RTRIG_1(CLK :=INPUT_VAR.I_LOTBOX_DETECT_1);
RTRIG_2(CLK :=INPUT_VAR.I_LOTBOX_DETECT_2);
RTRIG_3(CLK :=INPUT_VAR.I_LOTBOX_DETECT_3);
RTRIG_4(CLK :=INPUT_VAR.I_LOTBOX_DETECT_4);
(*
IF RTRIG_1.Q THEN
	IF QUEUE_INDEX_1 =0  THEN
		QUEUE_INDEX_1 :=1;
	ELSIF QUEUE_INDEX_2 =0 THEN
		QUEUE_INDEX_2 :=1;
	ELSIF QUEUE_INDEX_3 =0 THEN
		QUEUE_INDEX_3 :=1;
	ELSIF QUEUE_INDEX_4 =0 THEN
		QUEUE_INDEX_4 :=1;
	END_IF	
	INPUT_VAR.O_LOTBOX_CLAMP_ON_1:=TRUE;
	INPUT_VAR.O_LOTBOX_CLAMP_OFF_1:=FALSE;
ELSIF RTRIG_2.Q THEN
	IF QUEUE_INDEX_1 =0  THEN
		QUEUE_INDEX_1 :=2;
	ELSIF QUEUE_INDEX_2 =0 THEN
		QUEUE_INDEX_2 :=2;
	ELSIF QUEUE_INDEX_3 =0 THEN
		QUEUE_INDEX_3 :=2;
	ELSIF QUEUE_INDEX_4 =0 THEN
		QUEUE_INDEX_4 :=2;
	END_IF
	INPUT_VAR.O_LOTBOX_CLAMP_ON_2:=TRUE;
	INPUT_VAR.O_LOTBOX_CLAMP_OFF_2:=FALSE;
ELSIF RTRIG_3.Q THEN
	IF QUEUE_INDEX_1 =0  THEN
		QUEUE_INDEX_1 :=3;
	ELSIF QUEUE_INDEX_2 =0 THEN
		QUEUE_INDEX_2 :=3;
	ELSIF QUEUE_INDEX_3 =0 THEN
		QUEUE_INDEX_3 :=3;
	ELSIF QUEUE_INDEX_4 =0 THEN
		QUEUE_INDEX_4 :=3;
	END_IF	
	INPUT_VAR.O_LOTBOX_CLAMP_ON_3:=TRUE;
	INPUT_VAR.O_LOTBOX_CLAMP_OFF_3:=FALSE;
ELSIF RTRIG_4.Q THEN
	IF QUEUE_INDEX_1 =0  THEN
		QUEUE_INDEX_1 :=4;
	ELSIF QUEUE_INDEX_2 =0 THEN
		QUEUE_INDEX_2 :=4;
	ELSIF QUEUE_INDEX_3 =0 THEN
		QUEUE_INDEX_3 :=4;
	ELSIF QUEUE_INDEX_4 =0 THEN
		QUEUE_INDEX_4 :=4;
	END_IF	
	INPUT_VAR.O_LOTBOX_CLAMP_ON_4:=TRUE;
	INPUT_VAR.O_LOTBOX_CLAMP_OFF_4:=FALSE;	
END_IF

IF NOT INPUT_VAR.I_LOTBOX_DETECT_1 THEN
	QUEUE_INDEX_1 :=0;
END_IF
IF NOT INPUT_VAR.I_LOTBOX_DETECT_2 THEN
	QUEUE_INDEX_2 :=0;
END_IF
IF NOT INPUT_VAR.I_LOTBOX_DETECT_3 THEN
	QUEUE_INDEX_3 :=0;
END_IF
IF NOT INPUT_VAR.I_LOTBOX_DETECT_4 THEN
	QUEUE_INDEX_4 :=0;
END_IF

IF INPUT_VAR.I_LOTEND THEN
	INPUT_VAR.O_LOTBOX_CLAMP_ON_1:=FALSE;
	INPUT_VAR.O_LOTBOX_CLAMP_ON_2:=FALSE;
	INPUT_VAR.O_LOTBOX_CLAMP_ON_3:=FALSE;
	INPUT_VAR.O_LOTBOX_CLAMP_ON_4:=FALSE;
	INPUT_VAR.O_LOTBOX_CLAMP_OFF_1:=TRUE;
	INPUT_VAR.O_LOTBOX_CLAMP_OFF_2:=TRUE;
	INPUT_VAR.O_LOTBOX_CLAMP_OFF_3:=TRUE;
	INPUT_VAR.O_LOTBOX_CLAMP_OFF_4:=TRUE;
			
END_IF
*)	
 
(*
INPUT_VAR.O_STOPPER_TRANSFER_A:=TMR11.Q ;
INPUT_VAR.O_STOPPER_TRANSFER_B:=TMR12.Q ;

TMR14(IN:=INPUT_G6_VAR.I_G6_END_FUKUDA,PT:=T#10S);
IF NOT TMR14.Q AND INPUT_G6_VAR.I_G6_END_FUKUDA THEN
	TMR11(IN:=FALSE);
	TMR12(IN:=FALSE);
ELSE
	TMR11(IN:=INPUT_VAR.I_FUKUDA_TRANSFER_AT_FRONT_A,PT:=T#2S);	
	TMR12(IN:=INPUT_VAR.I_FUKUDA_TRANSFER_AT_FRONT_B,PT:=T#2S);

END_IF
 

 IF INPUT_G6_VAR.I_G6_END_FUKUDA AND NOT INPUT_VAR.ACTIVE_PROGRAM_CHANGE THEN
	INPUT_VAR.ACTIVE_PROGRAM:=INPUT_VAR.ACTIVE_PROGRAM+1;
	IF INPUT_VAR.ACTIVE_PROGRAM=3 THEN
		INPUT_VAR.ACTIVE_PROGRAM:=1;
	END_IF
	INPUT_VAR.ACTIVE_PROGRAM_CHANGE:=TRUE;
 END_IF

 COUNTER_1(CU:=INPUT_G6_VAR.I_G6_END_CYCLE,RESET:=INPUT_G6_VAR.O_G6_START,PV:=14);
IF COUNTER_1.CV =1 THEN
	INPUT_VAR.ACTIVE_PROGRAM_CHANGE:=FALSE;
END_IF
 
*)
PULS1(IN:=NOT PULS2.Q,PT:=T#0.5S);
PULS2(IN:=PULS1.Q,PT:=T#0.5S);
IF INPUT_VAR.I_LOTBOX_DETECT_1 THEN
	INPUT_VAR.O_LOT_BOX_INDICATOR_1:=PULS1.Q;
	LOTBOX_TEMPI1:=1;
ELSE
	INPUT_VAR.O_LOT_BOX_INDICATOR_1:=FALSE;
	LOTBOX_TEMPI1:=0;
END_IF

IF INPUT_VAR.I_LOTBOX_DETECT_2 THEN
	INPUT_VAR.O_LOT_BOX_INDICATOR_2:=PULS1.Q;
	LOTBOX_TEMPI2:=1;
	ELSE
	LOTBOX_TEMPI2:=0;
	INPUT_VAR.O_LOT_BOX_INDICATOR_2:=FALSE;
END_IF

IF INPUT_VAR.I_LOTBOX_DETECT_3 THEN
	INPUT_VAR.O_LOT_BOX_INDICATOR_3:=PULS1.Q;
	LOTBOX_TEMPI3:=1;
	ELSE
	INPUT_VAR.O_LOT_BOX_INDICATOR_3:=FALSE;
	LOTBOX_TEMPI3:=0;
END_IF

IF INPUT_VAR.I_LOTBOX_DETECT_4 THEN
	INPUT_VAR.O_LOT_BOX_INDICATOR_4:=PULS1.Q;
	LOTBOX_TEMPI4:=1;
	ELSE
	INPUT_VAR.O_LOT_BOX_INDICATOR_4:=FALSE;
	LOTBOX_TEMPI4:=0;
END_IF
LOTBOX_ACCI:=LOTBOX_TEMPI1 +LOTBOX_TEMPI2+LOTBOX_TEMPI3+LOTBOX_TEMPI4;

//IF LOTBOX_ACCI >=3 THEN
IF INPUT_G6_VAR.I_G6_MOTORON AND INDEXING_2_VAR.I_INDEXING_2_HOME AND  LOADER_RS4_VAR.I_LOADER_RS4_MOTORON AND INDEXING_1_VAR.I_INDEXING_1_HOME AND SORTER_RS4_VAR.I_SORTER_RS4_MOTORON AND TESTER_C8_VAR.I_C8_MOTORON THEN
	INPUT_VAR.O_TOWER_LAMP_GREEN :=TRUE;
	INPUT_VAR.O_TOWER_LAMP_RED :=FALSE;
	
	SORTER_VAR.O_TOWER_LAMP_GREEN :=TRUE;
	SORTER_VAR.O_TOWER_LAMP_RED :=FALSE;
ELSE
	INPUT_VAR.O_TOWER_LAMP_RED :=TRUE;
	INPUT_VAR.O_TOWER_LAMP_GREEN :=FALSE;
	
	SORTER_VAR.O_TOWER_LAMP_GREEN :=FALSE;
	SORTER_VAR.O_TOWER_LAMP_RED :=TRUE;
END_IF
IF LOTBOX_ACCI =2 OR LOTBOX_ACCI =1 THEN
	INPUT_VAR.O_TOWER_LAMP_YELLOW :=PULS1.Q;
END_IF
IF INPUT_VAR.ALARM1 THEN
	INPUT_VAR.O_TOWER_LAMP_YELLOW :=PULS1.Q;
	SORTER_VAR.O_TOWER_LAMP_YELLOW :=PULS1.Q;
	//INPUT_VAR.O_TOWER_LAMP_BUZZER :=TRUE;
END_IF

END_PROGRAM

// ---- POUs/FUKUDA/LOAD_FUKUDA.TcPOU
PROGRAM LOAD_FUKUDA
VAR_INPUT

END_VAR

VAR
	TMR_DELAY: TON;
	TMR1:TON;
	TMR_STOPPER_A: TON;
	TMR_STOPPER_B: TON;
	I_FUKUDA_TRANSFER_AT_BACK_BTHEN: INT;
	TMR_ALARM: TON;
END_VAR

IF 	INPUT_VAR.TRANSPORT_IDX=0 AND 	INPUT_VAR.STATION_LOAD_IDX=0 AND 	INPUT_VAR.JIG_LOAD_IDX =0 THEN
	INPUT_VAR.TRANSPORT_IDX:=	INPUT_VAR.I_CURRENT_TRANSACTION.TRANSPORT_INDEX;
	INPUT_VAR.STATION_LOAD_IDX:=INPUT_VAR.I_CURRENT_TRANSACTION.STATION_NUMBER_LOAD;
	INPUT_VAR.JIG_LOAD_IDX :=	INPUT_VAR.I_CURRENT_TRANSACTION.JIG_INDEX_LOAD;
ELSE
CASE INPUT_VAR.I_CASE OF
0: //standby near lotbox
	IF INPUT_VAR.ACTIVE_ID=6 THEN
		INPUT_VAR.ACTIVE_ID:=1;
	END_IF
	
	INPUT_VAR.TRANSPORT_IDX:=	INPUT_VAR.I_CURRENT_TRANSACTION.TRANSPORT_INDEX;
	INPUT_VAR.STATION_LOAD_IDX:=INPUT_VAR.I_CURRENT_TRANSACTION.STATION_NUMBER_LOAD;
	INPUT_VAR.JIG_LOAD_IDX :=	INPUT_VAR.I_CURRENT_TRANSACTION.JIG_INDEX_LOAD;
	CASE INPUT_VAR.TRANSPORT_IDX OF
		2 : FUKUDA_MOVE(STEP_DATA_1:=INPUT_VAR.STATION_LOAD_IDX,
				STEP_DATA_2:=3,
				STEP_DATA_3:=INPUT_VAR.JIG_LOAD_IDX,
				STEP_DATA_4:=0,
				STEP_DATA_5:=1);
				INPUT_VAR.O_STOPPER_TRANSFER_B:=FALSE;
		1 : FUKUDA_MOVE(STEP_DATA_1:=INPUT_VAR.STATION_LOAD_IDX,
				STEP_DATA_2:=3,
				STEP_DATA_3:=INPUT_VAR.JIG_LOAD_IDX,
				STEP_DATA_4:=1,
				STEP_DATA_5:=0);
				INPUT_VAR.O_STOPPER_TRANSFER_A:=FALSE;
	END_CASE			
	input_var.O_VACUUM_On:=FALSE;
	input_var.O_VACUUM_OFF:=FALSE;	
			
1: //standby near lotbox
	
	IF INPUT_VAR.ACTIVE_ID=6 THEN
		INPUT_VAR.ACTIVE_ID:=1;
	END_IF
		FUKUDA_MOVE(STEP_DATA_1:=INPUT_VAR.STATION_LOAD_IDX,
				STEP_DATA_2:=4,
				STEP_DATA_3:=INPUT_VAR.JIG_LOAD_IDX,
				STEP_DATA_4:=0,
				STEP_DATA_5:=0);

		CASE INPUT_VAR.TRANSPORT_IDX OF
		1:
			INPUT_VAR.I_LOADING_DONE_A:=FALSE;
		
		2:
			INPUT_VAR.I_LOADING_DONE_B:=FALSE;
	END_CASE
	
				
2://vacuum position 
	IF INPUT_VAR.ACTIVE_ID=6 THEN
		INPUT_VAR.ACTIVE_ID:=1;
	END_IF
	INPUT_VAR.I_CASE:=INPUT_VAR.I_CASE+1;
	(*FUKUDA_MOVE(STEP_DATA_1:=INPUT_VAR.I_CURRENT_TRANSACTION.STATION_NUMBER_LOAD,
				STEP_DATA_2:=4,
				STEP_DATA_3:=INPUT_VAR.I_CURRENT_TRANSACTION.JIG_INDEX_LOAD,
				STEP_DATA_4:=0,
				STEP_DATA_5:=0);
	IF INPUT_VAR.ACTIVE_ID=3 THEN
		input_var.O_VACUUM_ON:=TRUE;
		input_var.O_VACUUM_OFF:=FALSE;	
	END_IF
	*)

3://vacuum position 
	IF INPUT_VAR.ACTIVE_ID=6 THEN
		INPUT_VAR.ACTIVE_ID:=1; 
	END_IF
	//INPUT_VAR.I_CASE:=INPUT_VAR.I_CASE+1;
	//IF INPUT_VAR.O_VACUUM_ON THEN
		FUKUDA_MOVE(STEP_DATA_1:=INPUT_VAR.STATION_LOAD_IDX,
				STEP_DATA_2:=4,
				STEP_DATA_3:=INPUT_VAR.JIG_LOAD_IDX,
				STEP_DATA_4:=0,
				STEP_DATA_5:=0);
	//ELSE
		
	//END_IF
4://vacuum position 
	IF INPUT_VAR.ACTIVE_ID=6 THEN
		INPUT_VAR.ACTIVE_ID:=1;
	END_IF
	input_var.O_VACUUM_ON:=TRUE; 
	input_var.O_VACUUM_OFF:=FALSE;
	 
	//CHECK JIG FUKUDA PRESENCE			
	IF  input_var.O_VACUUM_ON THEN
		TMR1(IN:=INPUT_VAR.I_VACUUM_ON,PT:=T#3S);
	END_IF
	IF TMR1.Q  AND INPUT_VAR.I_VACUUM_ON THEN
		input_var.O_VACUUM_ON:=FALSE;
		INPUT_VAR.JIG_FUKUDA_PRESENCE :=FALSE;
		INPUT_VAR.I_CASE:=10;
	ELSE
				INPUT_VAR.JIG_FUKUDA_PRESENCE :=TRUE;	
				FUKUDA_MOVE(STEP_DATA_1:=INPUT_VAR.STATION_LOAD_IDX,
				STEP_DATA_2:=2,
				STEP_DATA_3:=INPUT_VAR.JIG_LOAD_IDX,
				STEP_DATA_4:=0,
				STEP_DATA_5:=0);
	END_IF
				
		

5://vacuum position 
	IF INPUT_VAR.ACTIVE_ID=6 THEN
		INPUT_VAR.ACTIVE_ID:=1;
	END_IF
	
	FUKUDA_MOVE(STEP_DATA_1:=8,
				STEP_DATA_2:=2,
				STEP_DATA_3:=INPUT_VAR.JIG_LOAD_IDX,
				STEP_DATA_4:=0,
				STEP_DATA_5:=0);
	
6://gripping position
	IF INPUT_VAR.ACTIVE_ID=6 THEN
		INPUT_VAR.ACTIVE_ID:=1;
	END_IF

	FUKUDA_MOVE(STEP_DATA_1:=INPUT_VAR.TRANSPORT_IDX+4,
				STEP_DATA_2:=2,
				STEP_DATA_3:=12,
				STEP_DATA_4:=0,
				STEP_DATA_5:=0);


7://placing onto fukuda transport
	IF INPUT_VAR.ACTIVE_ID=6 THEN
		INPUT_VAR.ACTIVE_ID:=1;
	END_IF
	FUKUDA_MOVE(STEP_DATA_1:=INPUT_VAR.TRANSPORT_IDX+4,
				STEP_DATA_2:=2,
				STEP_DATA_3:=11,
				STEP_DATA_4:=0,
				STEP_DATA_5:=0);

8://placing onto fukuda transport
	IF INPUT_VAR.ACTIVE_ID=6 THEN
		INPUT_VAR.ACTIVE_ID:=1;
	END_IF
	
	FUKUDA_MOVE(STEP_DATA_1:=INPUT_VAR.TRANSPORT_IDX+4,
				STEP_DATA_2:=2,
				STEP_DATA_3:=11,
				STEP_DATA_4:=0,
				STEP_DATA_5:=0);
	(*IF INPUT_VAR.ACTIVE_ID=3 THEN
		input_var.O_VACUUM_On:=FALSE;
		input_var.O_VACUUM_OFF:=TRUE;	
	END_IF
	*)
	
9://homing
	IF INPUT_VAR.ACTIVE_ID=6 THEN
		INPUT_VAR.ACTIVE_ID:=1;
	END_IF
	IF INPUT_VAR.I_VACUUM_ON THEN
		FUKUDA_MOVE(STEP_DATA_1:=INPUT_VAR.TRANSPORT_IDX+4,
				STEP_DATA_2:=1,
				STEP_DATA_3:=13,//11
				STEP_DATA_4:=0,
				STEP_DATA_5:=0);
	ELSE
		input_var.O_VACUUM_On:=FALSE;
		input_var.O_VACUUM_OFF:=TRUE;
	END_IF	
				
10://pusH fukuda transport
	IF INPUT_VAR.ACTIVE_ID=6 THEN
		INPUT_VAR.ACTIVE_ID:=1;
	END_IF
	input_var.O_VACUUM_On:=FALSE;
	input_var.O_VACUUM_OFF:=TRUE;
	CASE INPUT_VAR.TRANSPORT_IDX OF
		2 :
			//IF NOT INPUT_VAR.I_FUKUDA_TRANSFER_AT_FRONT_B   THEN
				FUKUDA_MOVE(STEP_DATA_1:=0,
				STEP_DATA_2:=0,
				STEP_DATA_3:=0,
				STEP_DATA_4:=0,
				STEP_DATA_5:=2);
			//END_IF
				 
		1 : 
			//IF NOT INPUT_VAR.I_FUKUDA_TRANSFER_AT_FRONT_A  THEN
				FUKUDA_MOVE(STEP_DATA_1:=0,
				STEP_DATA_2:=0,
				STEP_DATA_3:=0,
				STEP_DATA_4:=2,
				STEP_DATA_5:=0);
			//END_IF
	END_CASE			 
11:
		input_var.O_VACUUM_On:=FALSE;
		input_var.O_VACUUM_OFF:=FALSE;
		CASE INPUT_VAR.TRANSPORT_IDX OF
		1:	
			TMR_ALARM(IN:= NOT INPUT_VAR.I_FUKUDA_TRANSFER_AT_FRONT_A,PT:=T#50S);
			IF INPUT_VAR.I_FUKUDA_TRANSFER_AT_FRONT_A THEN
				TMR_STOPPER_A(IN:=TRUE,PT:=T#0.8S);
				IF TMR_STOPPER_A.Q THEN 
					TMR_ALARM(IN:=FALSE);
					INPUT_VAR.O_STOPPER_TRANSFER_A:=TRUE;
					INPUT_VAR.I_LOADING_DONE_A:=TRUE;
					TMR1(IN:=FALSE);
					TMR_DELAY(IN:=FALSE);
					input_var.O_VACUUM_On:=FALSE;
					input_var.O_VACUUM_OFF:=TRUE;
					FLAG_VAR.ALLOW_EXECUTE_LOAD_FUKUDA:=FALSE;
					INPUT_G6_VAR.I_G6_ENABLE:=TRUE;
					INPUT_VAR.I_CASE:=100;
				END_IF
				
			ELSE
				TMR_STOPPER_A(IN:=FALSE);
				FUKUDA_MOVE(STEP_DATA_1:=0,
				STEP_DATA_2:=0,
				STEP_DATA_3:=0,
				STEP_DATA_4:=2,
				STEP_DATA_5:=0);
			END_IF 
			
			2:
				TMR_ALARM(IN:= NOT INPUT_VAR.I_FUKUDA_TRANSFER_AT_FRONT_B,PT:=T#50S);
			IF INPUT_VAR.I_FUKUDA_TRANSFER_AT_FRONT_B THEN
				
				TMR_STOPPER_B(IN:=TRUE,PT:=T#0.8S);
				IF TMR_STOPPER_B.Q THEN
					TMR_ALARM(IN:=FALSE);
					INPUT_VAR.O_STOPPER_TRANSFER_B:=TRUE;	
					INPUT_VAR.I_LOADING_DONE_B:=TRUE;
					TMR1(IN:=FALSE);
					TMR_DELAY(IN:=FALSE);
					input_var.O_VACUUM_On:=FALSE;
					input_var.O_VACUUM_OFF:=TRUE;
					FLAG_VAR.ALLOW_EXECUTE_LOAD_FUKUDA:=FALSE;
					INPUT_G6_VAR.I_G6_ENABLE:=TRUE;
					INPUT_VAR.I_CASE:=100;
				END_IF
			ELSE
				TMR_STOPPER_B(IN:=FALSE);
				FUKUDA_MOVE(STEP_DATA_1:=0,
				STEP_DATA_2:=0,
				STEP_DATA_3:=0,
				STEP_DATA_4:=0,
				STEP_DATA_5:=2);
			END_IF
			
	END_CASE 
	IF TMR_ALARM.Q THEN
					INPUT_VAR.I_LOADING_DONE_B:=FALSE;
					TMR1(IN:=FALSE);
					TMR_DELAY(IN:=FALSE);
					input_var.O_VACUUM_On:=FALSE;
					input_var.O_VACUUM_OFF:=FALSE;
					FLAG_VAR.ALLOW_EXECUTE_LOAD_FUKUDA:=FALSE;
					INPUT_VAR.I_CASE:=100;
	END_IF
100:
	
	FLAG_VAR.ALLOW_EXECUTE_LOAD_FUKUDA:=FALSE;								
								
END_CASE 
END_IF

END_PROGRAM

// ---- POUs/FUKUDA/RETURN_FUKUDA.TcPOU
PROGRAM RETURN_FUKUDA
VAR_INPUT

END_VAR

VAR
	TMR_DELAY: TON;
END_VAR

IF 	INPUT_VAR.TRANSPORT_IDX=0 AND 	INPUT_VAR.STATION_RETURN_IDX=0 AND 	INPUT_VAR.JIG_RETURN_IDX =0 THEN
	INPUT_VAR.TRANSPORT_IDX:=	INPUT_VAR.I_CURRENT_TRANSACTION.TRANSPORT_INDEX;
	INPUT_VAR.STATION_RETURN_IDX:=INPUT_VAR.I_CURRENT_TRANSACTION.STATION_NUMBER_RETURN;
	INPUT_VAR.JIG_RETURN_IDX :=	INPUT_VAR.I_CURRENT_TRANSACTION.JIG_INDEX_RETURN;
ELSE
CASE INPUT_VAR.I_CASE OF
0: //standby near lotbox
	IF INPUT_VAR.ACTIVE_ID=6 THEN
		INPUT_VAR.ACTIVE_ID:=1;
	END_IF
	
	INPUT_VAR.TRANSPORT_IDX:=	INPUT_VAR.I_CURRENT_TRANSACTION.TRANSPORT_INDEX;
	INPUT_VAR.STATION_RETURN_IDX:=INPUT_VAR.I_CURRENT_TRANSACTION.STATION_NUMBER_RETURN;
	INPUT_VAR.JIG_RETURN_IDX :=	INPUT_VAR.I_CURRENT_TRANSACTION.JIG_INDEX_RETURN;

	CASE INPUT_VAR.TRANSPORT_IDX OF
		2 : 
			INPUT_VAR.O_STOPPER_TRANSFER_B:=FALSE;			
			FUKUDA_MOVE(STEP_DATA_1:=3,
				STEP_DATA_2:=1,
				STEP_DATA_3:=12,
				STEP_DATA_4:=0,
				STEP_DATA_5:=1);
				INPUT_VAR.O_STOPPER_TRANSFER_B:=FALSE;
		1 : 
			INPUT_VAR.O_STOPPER_TRANSFER_A:=FALSE;
			FUKUDA_MOVE(STEP_DATA_1:=3,
				STEP_DATA_2:=1,
				STEP_DATA_3:=12,
				STEP_DATA_4:=1,
				STEP_DATA_5:=0);
				INPUT_VAR.O_STOPPER_TRANSFER_A:=FALSE;
	END_CASE			
	input_var.O_VACUUM_On:=FALSE;
	input_var.O_VACUUM_OFF:=FALSE;	
	TMR_DELAY(IN:=FALSE);

1://ready for picking up
	IF INPUT_VAR.ACTIVE_ID=6 THEN
		INPUT_VAR.ACTIVE_ID:=1;
	END_IF

		CASE INPUT_VAR.TRANSPORT_IDX OF
		1:
			INPUT_VAR.I_RETURN_DONE_A:=FALSE;
		
		2:
			INPUT_VAR.I_RETURN_DONE_B:=FALSE;
	END_CASE
	FUKUDA_MOVE(STEP_DATA_1:=3,
				STEP_DATA_2:=1,
				STEP_DATA_3:=13,
				STEP_DATA_4:=0,
				STEP_DATA_5:=0);	
			
2://ready for picking up
	IF INPUT_VAR.ACTIVE_ID=6 THEN
		INPUT_VAR.ACTIVE_ID:=1;
	END_IF

	CASE INPUT_VAR.TRANSPORT_IDX OF
	1:		
		IF INPUT_VAR.I_FUKUDA_TRANSFER_AT_BACK_A THEN
		FUKUDA_MOVE(STEP_DATA_1:=INPUT_VAR.TRANSPORT_IDX+4,
				STEP_DATA_2:=1,
				STEP_DATA_3:=11,
				STEP_DATA_4:=0,
				STEP_DATA_5:=0);
		END_IF
	2:
		IF INPUT_VAR.I_FUKUDA_TRANSFER_AT_BACK_B THEN
		FUKUDA_MOVE(STEP_DATA_1:=INPUT_VAR.TRANSPORT_IDX+4,
				STEP_DATA_2:=1,
				STEP_DATA_3:=11,
				STEP_DATA_4:=0,
				STEP_DATA_5:=0);
	END_IF
	END_CASE
	
		
3://placing onto fukuda transport
	IF INPUT_VAR.ACTIVE_ID=6 THEN
		INPUT_VAR.ACTIVE_ID:=1;
	END_IF

	FUKUDA_MOVE(STEP_DATA_1:=INPUT_VAR.TRANSPORT_IDX+4,
				STEP_DATA_2:=2,
				STEP_DATA_3:=11,
				STEP_DATA_4:=0,
				STEP_DATA_5:=0);
	
4://ready for picking up
	IF INPUT_VAR.ACTIVE_ID=6 THEN
		INPUT_VAR.ACTIVE_ID:=1;
	END_IF
	
	FUKUDA_MOVE(STEP_DATA_1:=INPUT_VAR.TRANSPORT_IDX+4,
				STEP_DATA_2:=6,
				STEP_DATA_3:=11,
				STEP_DATA_4:=0,
				STEP_DATA_5:=0);

5://gripping position
	IF INPUT_VAR.ACTIVE_ID=6 THEN
		INPUT_VAR.ACTIVE_ID:=1;
	END_IF
	
	IF NOT input_var.I_VACUUM_On THEN
		FUKUDA_MOVE(STEP_DATA_1:=INPUT_VAR.TRANSPORT_IDX+4,
				STEP_DATA_2:=2,
				STEP_DATA_3:=12,
				STEP_DATA_4:=0,
				STEP_DATA_5:=0);
	ELSE
		input_var.O_VACUUM_On:=TRUE;
		input_var.O_VACUUM_OFF:=FALSE;
	END_IF
	
				
6://vacuum position 
	IF INPUT_VAR.ACTIVE_ID=6 THEN
		INPUT_VAR.ACTIVE_ID:=1;
	END_IF
	
	FUKUDA_MOVE(STEP_DATA_1:=INPUT_VAR.STATION_RETURN_IDX,
				STEP_DATA_2:=3,
				STEP_DATA_3:=INPUT_VAR.JIG_RETURN_IDX,
				STEP_DATA_4:=0,
				STEP_DATA_5:=0);
				
7://vacuum position 
	IF INPUT_VAR.ACTIVE_ID=6 THEN
		INPUT_VAR.ACTIVE_ID:=1;
	END_IF
	TMR_DELAY(IN:=TRUE,PT:=T#1S);
	IF TMR_DELAY.Q THEN
			FUKUDA_MOVE(STEP_DATA_1:=INPUT_VAR.STATION_RETURN_IDX,
				STEP_DATA_2:=3,
				STEP_DATA_3:=14,
				STEP_DATA_4:=0,
				STEP_DATA_5:=0);
	END_IF
				
8://vacuum position 
	IF INPUT_VAR.ACTIVE_ID=6 THEN
		INPUT_VAR.ACTIVE_ID:=1;
	END_IF
	TMR_DELAY(IN:=FALSE);
	FUKUDA_MOVE(STEP_DATA_1:=INPUT_VAR.STATION_RETURN_IDX,
				STEP_DATA_2:=7,
				STEP_DATA_3:=16,
				STEP_DATA_4:=0,
				STEP_DATA_5:=0);
				
9://vacuum position 
	IF INPUT_VAR.ACTIVE_ID=6 THEN
		INPUT_VAR.ACTIVE_ID:=1;
	END_IF
	
	FUKUDA_MOVE(STEP_DATA_1:=INPUT_VAR.STATION_RETURN_IDX,
				STEP_DATA_2:=8,
				STEP_DATA_3:=INPUT_VAR.JIG_RETURN_IDX,
				STEP_DATA_4:=0,
				STEP_DATA_5:=0);
10: //standby near lotbox
	
	IF INPUT_VAR.ACTIVE_ID=6 THEN
		INPUT_VAR.ACTIVE_ID:=1;
	END_IF

	IF input_var.I_VACUUM_ON THEN
		FUKUDA_MOVE(STEP_DATA_1:=INPUT_VAR.STATION_RETURN_IDX,
				STEP_DATA_2:=4,
				STEP_DATA_3:=INPUT_VAR.JIG_RETURN_IDX,
				STEP_DATA_4:=0,
				STEP_DATA_5:=0);
	ELSE
		input_var.O_VACUUM_ON:=FALSE;
		input_var.O_VACUUM_OFF:=TRUE;			
	END_IF
	
				
11://vacuum position 
	IF INPUT_VAR.ACTIVE_ID=6 THEN
		INPUT_VAR.ACTIVE_ID:=1;
	END_IF
	FUKUDA_MOVE(STEP_DATA_1:=INPUT_VAR.STATION_RETURN_IDX,
				STEP_DATA_2:=1,
				STEP_DATA_3:=INPUT_VAR.JIG_RETURN_IDX,
				STEP_DATA_4:=0,
				STEP_DATA_5:=0);
	IF INPUT_VAR.ACTIVE_ID=3 THEN
		input_var.O_VACUUM_ON:=FALSE;
		input_var.O_VACUUM_OFF:=FALSE;	
	END_IF
	
12://vacuum position 
	IF INPUT_VAR.ACTIVE_ID=6 THEN
		INPUT_VAR.ACTIVE_ID:=1;
	END_IF
	FUKUDA_MOVE(STEP_DATA_1:=0,
				STEP_DATA_2:=1,
				STEP_DATA_3:=4,
				STEP_DATA_4:=0,
				STEP_DATA_5:=0);				
		
100:
	
	input_var.O_VACUUM_On:=FALSE;
	input_var.O_VACUUM_OFF:=FALSE;
END_CASE 
END_IF
IF INPUT_VAR.I_CASE=13 THEN
			CASE INPUT_VAR.TRANSPORT_IDX OF
		1:
			INPUT_VAR.I_RETURN_DONE_A:=TRUE;
		
		2:
			INPUT_VAR.I_RETURN_DONE_B:=TRUE;
	END_CASE
	IF INPUT_VAR.I_RETURN_DONE_A OR INPUT_VAR.I_RETURN_DONE_B THEN
		FLAG_VAR.ALLOW_EXECUTE_RETURN_FUKUDA:=FALSE;
		INPUT_VAR.I_CASE:=100;
	END_IF
END_IF

END_PROGRAM

// ---- POUs/FUKUDA/LOAD_FUKUDA_1.TcPOU
PROGRAM LOAD_FUKUDA_1
VAR_INPUT

END_VAR

VAR
	TMR_DELAY: TON;
	TMR1:TON;
END_VAR

CASE INPUT_VAR.I_CASE OF
0: //standby near lotbox
	IF INPUT_VAR.ACTIVE_ID=6 THEN
		INPUT_VAR.ACTIVE_ID:=1;
	END_IF
	CASE INPUT_VAR.I_CURRENT_TRANSACTION.TRANSPORT_INDEX OF
		2 : FUKUDA_MOVE(STEP_DATA_1:=INPUT_VAR.I_CURRENT_TRANSACTION.STATION_NUMBER_LOAD,
				STEP_DATA_2:=3,
				STEP_DATA_3:=INPUT_VAR.I_CURRENT_TRANSACTION.JIG_INDEX_LOAD,
				STEP_DATA_4:=0,
				STEP_DATA_5:=1);
		1 : FUKUDA_MOVE(STEP_DATA_1:=INPUT_VAR.I_CURRENT_TRANSACTION.STATION_NUMBER_LOAD,
				STEP_DATA_2:=3,
				STEP_DATA_3:=INPUT_VAR.I_CURRENT_TRANSACTION.JIG_INDEX_LOAD,
				STEP_DATA_4:=1,
				STEP_DATA_5:=0);
				
	input_var.O_VACUUM_On:=FALSE;
	input_var.O_VACUUM_OFF:=FALSE;	
	TMR_DELAY(IN:=FALSE);

	END_CASE
				
1: //standby near lotbox
	
	IF INPUT_VAR.ACTIVE_ID=6 THEN
		INPUT_VAR.ACTIVE_ID:=1;
	END_IF
		FUKUDA_MOVE(STEP_DATA_1:=INPUT_VAR.I_CURRENT_TRANSACTION.STATION_NUMBER_LOAD,
				STEP_DATA_2:=4,
				STEP_DATA_3:=INPUT_VAR.I_CURRENT_TRANSACTION.JIG_INDEX_LOAD,
				STEP_DATA_4:=0,
				STEP_DATA_5:=0);

		CASE INPUT_VAR.I_CURRENT_TRANSACTION.TRANSPORT_INDEX OF
		1:
			INPUT_VAR.I_LOADING_DONE_A:=FALSE;
		
		2:
			INPUT_VAR.I_LOADING_DONE_B:=FALSE;
	END_CASE

		
				
2://vacuum position 
	IF INPUT_VAR.ACTIVE_ID=6 THEN
		INPUT_VAR.ACTIVE_ID:=1;
	END_IF
	FUKUDA_MOVE(STEP_DATA_1:=INPUT_VAR.I_CURRENT_TRANSACTION.STATION_NUMBER_LOAD,
				STEP_DATA_2:=4,
				STEP_DATA_3:=INPUT_VAR.I_CURRENT_TRANSACTION.JIG_INDEX_LOAD,
				STEP_DATA_4:=0,
				STEP_DATA_5:=0);
	IF INPUT_VAR.ACTIVE_ID=3 THEN
		input_var.O_VACUUM_ON:=TRUE;
		input_var.O_VACUUM_OFF:=FALSE;	
	END_IF

3://vacuum position 
	IF INPUT_VAR.ACTIVE_ID=6 THEN
		INPUT_VAR.ACTIVE_ID:=1; 
	END_IF
	FUKUDA_MOVE(STEP_DATA_1:=INPUT_VAR.I_CURRENT_TRANSACTION.STATION_NUMBER_LOAD,
				STEP_DATA_2:=4,
				STEP_DATA_3:=INPUT_VAR.I_CURRENT_TRANSACTION.JIG_INDEX_LOAD,
				STEP_DATA_4:=0,
				STEP_DATA_5:=0);
	
 		
//CHECK JIG FUKUDA PRESENCE			
	IF  input_var.O_VACUUM_ON THEN
		TMR1(IN:=TRUE,PT:=T#2S);
		IF TMR1.Q THEN
			IF NOT INPUT_VAR.I_VACUUM_ON AND input_var.O_VACUUM_ON THEN
				INPUT_VAR.JIG_FUKUDA_PRESENCE :=TRUE;
			ELSE
				INPUT_VAR.JIG_FUKUDA_PRESENCE :=FALSE;	
				FUKUDA_MOVE(STEP_DATA_1:=INPUT_VAR.I_CURRENT_TRANSACTION.STATION_NUMBER_LOAD,
				STEP_DATA_2:=2,
				STEP_DATA_3:=INPUT_VAR.I_CURRENT_TRANSACTION.JIG_INDEX_LOAD,
				STEP_DATA_4:=0,
				STEP_DATA_5:=0);
				
				FUKUDA_MOVE(STEP_DATA_1:=INPUT_VAR.I_CURRENT_TRANSACTION.STATION_NUMBER_LOAD,
				STEP_DATA_2:=1,
				STEP_DATA_3:=INPUT_VAR.I_CURRENT_TRANSACTION.JIG_INDEX_LOAD,
				STEP_DATA_4:=0,
				STEP_DATA_5:=0);
			input_var.O_VACUUM_ON:=FALSE;
			input_var.O_VACUUM_OFF:=FALSE;
			TMR_DELAY(IN:=TRUE,PT:=T#2.5S);
		
			IF TMR_DELAY.Q THEN
				FLAG_VAR.ALLOW_EXECUTE_LOAD_FUKUDA:=FALSE;
				INPUT_VAR.I_CURRENT_TRANSACTION.JIG_INDEX_LOAD:=INPUT_VAR.I_CURRENT_TRANSACTION.JIG_INDEX_LOAD+0;
				INPUT_VAR.I_CASE:=0;
			END_IF
		END_IF
	ELSE
		TMR1(IN:=FALSE);	
	END_IF 
		
				//INPUT_VAR.JIG_FUKUDA_PRESENCE :=TRUE;
				//IF INPUT_VAR.I_CURRENT_TRANSACTION.JIG_INDEX_LOAD >=11 THEN
					//INPUT_VAR.I_CASE:=100;
			
				//FLAG_VAR.ALLOW_EXECUTE_LOAD_FUKUDA:=FALSE;
				//INPUT_VAR.I_CASE:=0;
				//INPUT_VAR.I_CURRENT_TRANSACTION.JIG_INDEX_LOAD:=1 ;
					//ELSE
						
				//END_IF
				
				//TMR_DELAY(IN:=FALSE);
				//LOAD_FUKUDA();
				//FLAG_VAR.ALLOW_EXECUTE_LOAD_FUKUDA:=FALSE;
	
	END_IF
 
	
4://vacuum position 
	IF INPUT_VAR.ACTIVE_ID=6 THEN
		INPUT_VAR.ACTIVE_ID:=1;
	END_IF
	
	FUKUDA_MOVE(STEP_DATA_1:=7,
				STEP_DATA_2:=4,
				STEP_DATA_3:=INPUT_VAR.I_CURRENT_TRANSACTION.JIG_INDEX_LOAD,
				STEP_DATA_4:=0,
				STEP_DATA_5:=0);
				

5://vacuum position 
	IF INPUT_VAR.ACTIVE_ID=6 THEN
		INPUT_VAR.ACTIVE_ID:=1;
	END_IF
	
	FUKUDA_MOVE(STEP_DATA_1:=8,
				STEP_DATA_2:=2,
				STEP_DATA_3:=INPUT_VAR.I_CURRENT_TRANSACTION.JIG_INDEX_LOAD,
				STEP_DATA_4:=0,
				STEP_DATA_5:=0);
	
6://gripping position
	IF INPUT_VAR.ACTIVE_ID=6 THEN
		INPUT_VAR.ACTIVE_ID:=1;
	END_IF

	FUKUDA_MOVE(STEP_DATA_1:=INPUT_VAR.I_CURRENT_TRANSACTION.TRANSPORT_INDEX+4,
				STEP_DATA_2:=2,
				STEP_DATA_3:=12,
				STEP_DATA_4:=0,
				STEP_DATA_5:=0);


7://placing onto fukuda transport
	IF INPUT_VAR.ACTIVE_ID=6 THEN
		INPUT_VAR.ACTIVE_ID:=1;
	END_IF
	FUKUDA_MOVE(STEP_DATA_1:=INPUT_VAR.I_CURRENT_TRANSACTION.TRANSPORT_INDEX+4,
				STEP_DATA_2:=2,
				STEP_DATA_3:=11,
				STEP_DATA_4:=0,
				STEP_DATA_5:=0);

8://placing onto fukuda transport
	IF INPUT_VAR.ACTIVE_ID=6 THEN
		INPUT_VAR.ACTIVE_ID:=1;
	END_IF
	
	FUKUDA_MOVE(STEP_DATA_1:=INPUT_VAR.I_CURRENT_TRANSACTION.TRANSPORT_INDEX+4,
				STEP_DATA_2:=2,
				STEP_DATA_3:=11,
				STEP_DATA_4:=0,
				STEP_DATA_5:=0);
	IF INPUT_VAR.ACTIVE_ID=3 THEN
		input_var.O_VACUUM_On:=FALSE;
		input_var.O_VACUUM_OFF:=TRUE;	
	END_IF

	
9://homing
	IF INPUT_VAR.ACTIVE_ID=6 THEN
		INPUT_VAR.ACTIVE_ID:=1;
	END_IF
	
	FUKUDA_MOVE(STEP_DATA_1:=INPUT_VAR.I_CURRENT_TRANSACTION.TRANSPORT_INDEX+4,
				STEP_DATA_2:=1,
				STEP_DATA_3:=11,
				STEP_DATA_4:=0,
				STEP_DATA_5:=0);
			
				
10://pusH fukuda transport
	IF INPUT_VAR.ACTIVE_ID=6 THEN
		INPUT_VAR.ACTIVE_ID:=1;
	END_IF
	input_var.O_VACUUM_OFF:=FALSE;
	CASE INPUT_VAR.I_CURRENT_TRANSACTION.TRANSPORT_INDEX OF
		2 : FUKUDA_MOVE(STEP_DATA_1:=0,
				STEP_DATA_2:=0,
				STEP_DATA_3:=0,
				STEP_DATA_4:=0,
				STEP_DATA_5:=2);
		1 : FUKUDA_MOVE(STEP_DATA_1:=0,
				STEP_DATA_2:=0,
				STEP_DATA_3:=0,
				STEP_DATA_4:=2,
				STEP_DATA_5:=0);
	END_CASE			 

100:

	input_var.O_VACUUM_On:=FALSE;
	input_var.O_VACUUM_OFF:=FALSE;	
	
END_CASE 
IF INPUT_VAR.I_CASE=11 THEN
			CASE INPUT_VAR.I_CURRENT_TRANSACTION.TRANSPORT_INDEX OF
		1:	
			IF INPUT_VAR.I_FUKUDA_TRANSFER_AT_FRONT_A THEN
				INPUT_VAR.I_LOADING_DONE_A:=TRUE;
				IF  INPUT_VAR.I_LOADING_DONE_A THEN
					FLAG_VAR.ALLOW_EXECUTE_LOAD_FUKUDA:=FALSE;			
					INPUT_VAR.I_CASE:=100;
				END_IF
			END_IF
			
				2:
			IF INPUT_VAR.I_FUKUDA_TRANSFER_AT_FRONT_B THEN
				INPUT_VAR.I_LOADING_DONE_B:=TRUE;
				IF  INPUT_VAR.I_LOADING_DONE_B THEN
					FLAG_VAR.ALLOW_EXECUTE_LOAD_FUKUDA:=FALSE;			
					INPUT_VAR.I_CASE:=100;
				END_IF
			END_IF
			
	END_CASE

END_IF

END_PROGRAM

// ---- POUs/LASER/LASER_MOVE.TcPOU
PROGRAM LASER_MOVE
//FUNCTION LASER_MOVE : BOOL
VAR_INPUT
	STEP_DATA_1: BYTE;
	STEP_DATA_2: BYTE;
	STEP_DATA_3: BYTE;
	STEP_DATA_4: BYTE;
	STEP_DATA_5: BYTE;

END_VAR

VAR
	
	(*
DataWordInput1 AT %IB232 : ARRAY [0..15] OF WORD; 
DataWordInput2 AT %IB264 : ARRAY [16..31] OF WORD;
DataWordInput3 AT %IB264 : ARRAY [32..47] OF WORD; 
DataWordInput4 AT %IB296 : ARRAY [48..56] OF WORD; 
DataWordOutput1 AT %QB232 : ARRAY [0..15] OF WORD; 
DataWordOutput2 AT %QB264 : ARRAY [16..31] OF WORD; 
DataWordOutput3 AT %QB296 : ARRAY [32..47] OF WORD; 
DataWordOutput4 AT %QB328 : ARRAY [48..56] OF WORD; 

DataWordInput1 AT %IB100 : ARRAY [0..15] OF WORD; 
DataWordInput2 AT %IB132 : ARRAY [16..31] OF WORD; 
DataWordInput3 AT %IB164 : ARRAY [32..47] OF WORD; 
DataWordInput4 AT %IB196 : ARRAY [48..56] OF WORD; 
DataWordOutput1 AT %QB100 : ARRAY [0..15] OF WORD; 
DataWordOutput2 AT %QB132 : ARRAY [16..31] OF WORD; 
DataWordOutput3 AT %QB164 : ARRAY [32..47] OF WORD; 
DataWordOutput4 AT %QB196 : ARRAY [48..56] OF WORD; 
	*)
	Gateway_Q0_MODE_COMMAND_0 AT %QX232.0 : BOOL ;
	Gateway_Q0_MODE_COMMAND_1 AT %QX232.1 : BOOL ;
	Gateway_Q0_RESET AT %QX232.4 : BOOL;
	Gateway_Q0_RESTART AT %QX232.5 : BOOL;
	Gateway_Q0_STOP AT %QX232.7 : BOOL;
	Gateway_Q1_0 AT %QX233.0 : BOOL;
	Gateway_Q1_1 AT %QX233.1 : BOOL;
	Gateway_Q1_2 AT %QX233.2 : BOOL;
	Gateway_Q1_3 AT %QX233.3 : BOOL;
	Gateway_Q1_4 AT %QX233.4 : BOOL;
	Gateway_Gateway_Unit_2_Status AT %QB234 : BYTE;
	Gateway_Q3_0 AT %QX235.0 : BOOL;
	Gateway_Q3_1 AT %QX235.1 : BOOL;
	Gateway_Q3_2 AT %QX235.2 : BOOL;
	Gateway_Q3_3 AT %QX235.3 : BOOL;	
	

	ID1_StepData AT %QB246 : BYTE;
	ID1_Hold AT %QX247.0 : BOOL;
	ID1_SVON AT %QX247.1 : BOOL;
	ID1_Drive AT %QX247.2 : BOOL;
	ID1_Reset AT %QX247.3 : BOOL;
	ID1_Setup AT %QX247.4 : BOOL;
	

	ID2_StepData AT %QB266 : BYTE;
	ID2_Hold AT %QX267.0 : BOOL;
	ID2_SVON AT %QX267.1 : BOOL;
	ID2_Drive AT %QX267.2 : BOOL;
	ID2_Reset AT %QX267.3 : BOOL;
	ID2_Setup AT %QX267.4 : BOOL;


	ID3_StepData AT %QB286 : BYTE;
	ID3_Hold AT %QX287.0 : BOOL;
	ID3_SVON AT %QX287.1 : BOOL;
	ID3_Drive AT %QX287.2 : BOOL;
	ID3_Reset AT %QX287.3 : BOOL;
	ID3_Setup AT %QX287.4 : BOOL;
	
	
	ID4_StepData AT %QB306 : BYTE;
	ID4_Hold AT %QX307.0 : BOOL;
	ID4_SVON AT %QX307.1 : BOOL;
	ID4_Drive AT %QX307.2 : BOOL;
	ID4_Reset AT %QX307.3 : BOOL;
	ID4_Setup AT %QX307.4 : BOOL;
	

	ID5_StepData AT %QB326 : BYTE;
	ID5_Hold AT %QX327.0 : BOOL;
	ID5_SVON AT %QX327.1 : BOOL;
	ID5_Drive AT %QX327.2 : BOOL;
	ID5_Reset AT %QX327.3 : BOOL;
	ID5_Setup AT %QX327.4 : BOOL;
	
	byte0 : BYTE;
	byte1 : BYTE;
	byte2 : BYTE;
	byte3 : BYTE;
	
	bit14_0 : BOOL;
	bit14_1 : BOOL;
	bit14_2 : BOOL;
	bit14_3 : BOOL;
	bit14_4 : BOOL;
	bit14_5 : BOOL;
	
	bit15_0 : BOOL;
	bit15_1 : BOOL;
	bit15_2 : BOOL;
	bit15_3 : BOOL;
	bit15_4 : BOOL; 
	
	bit34_0 : BOOL;
	bit34_1 : BOOL;
	bit34_2 : BOOL;
	bit34_3 : BOOL;
	bit34_4 : BOOL;
	bit34_5 : BOOL;
	
	bit35_0 : BOOL;
	bit35_1 : BOOL;
	bit35_2 : BOOL;
	bit35_3 : BOOL;
	bit35_4 : BOOL; 
	
	bit54_0 : BOOL;
	bit54_1 : BOOL;
	bit54_2 : BOOL;
	bit54_3 : BOOL;
	bit54_4 : BOOL;
	bit54_5 : BOOL;
	
	bit55_0 : BOOL;
	bit55_1 : BOOL;
	bit55_2 : BOOL;
	bit55_3 : BOOL;
	bit55_4 : BOOL; 
	
	bit74_0 : BOOL;
	bit74_1 : BOOL;
	bit74_2 : BOOL;
	bit74_3 : BOOL;
	bit74_4 : BOOL;
	bit74_5 : BOOL;
	
	bit75_0 : BOOL;
	bit75_1 : BOOL;
	bit75_2 : BOOL;
	bit75_3 : BOOL;
	bit75_4 : BOOL; 
	
	bit94_0 : BOOL;
	bit94_1 : BOOL;
	bit94_2 : BOOL;
	bit94_3 : BOOL;
	bit94_4 : BOOL;
	bit94_5 : BOOL;
	
	bit95_0 : BOOL;
	bit95_1 : BOOL;
	bit95_2 : BOOL;
	bit95_3 : BOOL;
	bit95_4 : BOOL; 	
	
	ID1_I0_MODE_COMMAND_0 AT %IX232.0 : BOOL :=0;
	ID1_I0_MODE_COMMAND_1 AT %IX232.1 : BOOL:=0;
	ID1_I0_READY AT %IX232.4 : BOOL;
	ID1_I0_ALARM AT %IX232.5 : BOOL;
	ID1_I0_INITIAL AT %IX232.6 : BOOL;
	ID1_I0_COMMUNICATING AT %IX232.7 : BOOL;
	ID1_I1_0 AT %IX233.0 : BOOL;
	ID1_I1_1 AT %IX233.1 : BOOL;
	ID1_I1_2 AT %IX233.2 : BOOL;
	ID1_I1_3 AT %IX233.3 : BOOL;
	ID1_I1_4 AT %IX233.4 : BOOL;
	ID1_I2_0 AT %IX234.0 : BOOL;
	ID1_I2_1 AT %IX234.1 : BOOL;
	ID1_I2_2 AT %IX234.2 : BOOL;
	ID1_I2_3 AT %IX234.3 : BOOL;
	ID1_I2_4 AT %IX234.4 : BOOL;

	ID1_I3_0 AT %IX235.0 : BOOL;
	ID1_I3_1 AT %IX235.1 : BOOL;
	
	ID1_I32_0 AT %IX264.0 : BOOL;
	ID1_I32_1 AT %IX264.1 : BOOL;
	ID1_I33_0 AT %IX265.0 : BOOL;
	ID1_I33_1 AT %IX265.1 : BOOL;
(*-----------------------------------------------------------*)

	iTest15: SINT;
	iTest16: SINT;
	
	bTest1 : BOOL;
	bTest2 : BOOL;
	bTest3 : BOOL;
	bTest4 : BOOL;
	bTest5 : BOOL;
	bTest6 : BOOL;
	bTest7 : BOOL;
	bTest8 : BOOL;
	bTest9 : BOOL;
	bTest10 : BOOL;
	bTest11 : BOOL;
	bTest12 : BOOL;
	bTest13 : BOOL;
	bTest14 : BOOL;
	
	StepData1 : BYTE;
	StepData2 : BYTE;
	StepData3 : BYTE;
	StepData4 : BYTE;
	StepData5 : BYTE;
	
	star :BOOL;
	hom : BOOL;

	reset: BOOL;
	
	ID1_ALARM AT%IX247.7 : BOOL;
	ID2_ALARM AT%IX267.7 : BOOL;
	ID3_ALARM AT%IX287.7 : BOOL;
	ID4_ALARM AT%IX307.7 : BOOL;
	ID5_ALARM AT%IX327.7 : BOOL;
	
	ID1_SVRE AT%IX247.1 : BOOL;
	ID2_SVRE AT%IX267.1 : BOOL;
	ID3_SVRE AT%IX287.1 : BOOL;
	ID4_SVRE AT%IX307.1 : BOOL;
	ID5_SVRE AT%IX327.1 : BOOL;
	
	ID1_INP AT%IX247.3 : BOOL;
	ID2_INP AT%IX267.3 : BOOL;
	ID3_INP AT%IX287.3 : BOOL;
	ID4_INP AT%IX307.3 : BOOL;
	ID5_INP AT%IX327.3 : BOOL;
	
	PROSES: STRING;
	STAGE: INT;
	
	PROCESS: INT;
	START_PROCESS: BOOL;
	STEP_DATAS: INT;
	PROCESS_DELAY: TIME :=T#300MS;
	LASER_RUNNING: BOOL :=FALSE;
	ACTIVE_STEPDATA : BYTE;
	//ACTIVE_ID: INT :=1;
	TMR1: TON;
	TMR2: TON;
	TMR3: TON;
	TMR4: TON;
	TMR5: TON;
	TMR6: TON;
	TMR10: Ton;
	TMR11: TON;
	TMR12: TON;
	TMR13: TON;
	TMR14: TON;
	TMR20: TON;
	TMR21: TON;
	TMR22: TON;
	TMR23: TON;
	TMR30: TON;
	TMR31: TON;
	TMR32: TON;
	TMR33: TON;
	TMR40: TON;
	TMR41: TON;
	TMR42: TON;
	TMR43: TON;
	TMR50: TON;
	TMR51: TON;
	TMR52: TON;
	TMR53: TON;
	
	
	TMR101: TON;
	TMR102: TON;
	TMR103: TON;
	TMR104: TON;
	TMR105: TON;
	TMR106: TON;
	ID5: INT;
	TMR7: Ton;
	TMR_RES_CARTSN: TOF;
	TMR_ACTIVATE_RESET: TON;
	TMR_RST: TON;
	TMR_RST1: TON;
	ID2_READY: BOOL;
	ID4_READY: BOOL;
	ID5_READY: BOOL;
END_VAR


PROCESS_DELAY:= T#400MS;
IF 	SORTER_VAR.ACTIVE_ID >=0 THEN
STEP_DATA_1:=STEP_DATA_1+1;

IF STEP_DATA_2>=5 THEN
	STEP_DATA_2:=STEP_DATA_2+1;
END_IF

STEP_DATA_3:=STEP_DATA_3+1;	
END_IF

IF NOT ID1_SVRE OR NOT ID2_SVRE OR NOT ID3_SVRE OR NOT ID4_SVRE OR NOT ID5_SVRE THEN
	TMR_RST(IN:=TRUE,PT:=T#10S);
	IF TMR_RST.Q THEN
		SORTER_VAR.O_RESET_CARTESSIAN:=TRUE;
		TMR_RST1(IN:=TRUE,PT:=T#1S);
		IF TMR_RST1.Q THEN
			SORTER_VAR.O_RESET_CARTESSIAN:=FALSE;
			TMR_RST(IN:=FALSE);
			TMR_RST1(IN:=FALSE);
			FLAG_VAR.ALLOW_EXECUTE_LOAD_LASER :=FALSE;
			FLAG_VAR.ALLOW_EXECUTE_RETURN_LASER:=FALSE;
			LASER_MOVE(STEP_DATA_1:=0,
				STEP_DATA_2:=0,
				STEP_DATA_3:=0,
				STEP_DATA_4:=0,
				STEP_DATA_5:=0);
		END_IF
	END_IF
ELSE
	SORTER_VAR.O_RESET_CARTESSIAN:=FALSE;
	TMR_RST(IN:=FALSE);
	TMR_RST1(IN:=FALSE);
END_IF
IF NOT SORTER_VAR.LASER_HOME THEN //LASER_running THEN
	IF  ID1_SVRE AND ID2_SVRE  AND  ID3_SVRE AND  ID4_SVRE AND  ID5_SVRE THEN
		TMR1(IN:=TRUE,PT:=T#0.5S);
		TMR4(IN:=TRUE,PT:=T#5S);
		TMR5(IN:=TRUE,PT:=T#5.5S);
		TMR6(IN:=TRUE,PT:=T#25S);
		
		IF ID2_SVRE THEN
			ID2_SETUP:=TRUE;
			IF ID2_INP THEN
				ID2_READY:=TRUE;
				IF ID3_SVRE THEN
					ID3_SETUP :=TRUE;
					IF ID3_INP THEN
						ID2_READY:=TRUE;
						IF ID1_SVRE THEN
							ID1_SETUP :=TRUE;
						ELSE
							ID1_SVON :=TRUE;	
						END_IF
					END_IF
				ELSE
					ID3_SVON :=TRUE;
				END_IF
			END_IF
		ELSE
			ID2_SVON :=TRUE;					
		END_IF
		(*
		IF ID1_SVRE THEN
			ID1_SETUP :=TMR5.Q;
		ELSE
			ID1_SVON :=TRUE;	
		END_IF

		IF ID2_SVRE THEN
			ID2_SETUP :=TMR1.Q;
		ELSE
			ID2_SVON :=TRUE;	
		END_IF
	
		IF ID3_SVRE THEN
		ID3_SETUP :=TMR4.Q;
		ELSE
			ID3_SVON :=TRUE;	
		END_IF
		*)
		CASE SORTER_VAR.I_CURRENT_TRANSACTION.TRANSPORT_INDEX OF
		1:
			TMR2(IN:=TRUE,PT:=T#1S);
			IF ID4_SVRE THEN
				ID4_SETUP :=TMR2.Q;
				IF ID4_INP THEN
					ID4_READY:=TRUE;
				END_IF
			ELSE
				ID4_SVON :=TRUE;	
			END_IF
		2:
			TMR3(IN:=TRUE,PT:=T#1.5S);
			IF ID5_SVRE THEN
				ID5_SETUP :=TMR3.Q;
				IF ID5_INP THEN
					ID5_READY:=TRUE;
				END_IF
			ELSE
				ID5_SVON :=TRUE;	
			END_IF
		END_CASE

	//IF TMR6.Q THEN
	IF ID1_INP AND ID2_INP AND ID3_INP AND (ID4_INP OR ID5_INP) THEN
		ID1_SETUP :=FALSE;
		ID2_SETUP :=FALSE;
		ID3_SETUP :=FALSE;
		ID4_SETUP :=FALSE;
		ID5_SETUP :=FALSE;
	
		TMR1(IN:=FALSE);
		TMR2(IN:=FALSE);
		TMR3(IN:=FALSE);
		TMR4(IN:=FALSE);
		TMR5(IN:=FALSE);
	//ACTIVE_ID:=1;
	//LASER_RUNNING:=TRUE;
		SORTER_VAR.LASER_HOME:=TRUE;
	END_IF
	
	ELSE
				
	ID1_SVON :=TRUE;
	ID2_SVON :=TRUE;
	ID3_SVON :=TRUE;
	ID4_SVON :=TRUE;
	ID5_SVON :=TRUE;

	END_IF
ELSE
	TMR6(IN:=FALSE);

	CASE SORTER_VAR.ACTIVE_ID OF
	0:
		//SORTER_VAR.I_LASER_RUNNING:=FALSE;
		SORTER_VAR.ACTIVE_ID:=6;
		IF 	FLAG_VAR.ALLOW_EXECUTE_LOAD_NG OR FLAG_VAR.ALLOW_EXECUTE_RETURN_NG THEN
			SORTER_VAR.I_NG_CASE:=SORTER_VAR.I_NG_CASE+1;
		ELSE
			SORTER_VAR.I_CASE:=SORTER_VAR.I_CASE+1;
		END_IF
	1:
		IF STEP_DATA_1 = 0 THEN
			SORTER_VAR.ACTIVE_ID:=2;
		ELSE
			IF ID1_ALARM THEN
				Reset := TRUE;
				TMR10(IN:=TRUE,PT:= PROCESS_DELAY);
				IF TMR10.Q THEN
					Reset := FALSE;
				END_IF
			ELSE
				ID1_StepData :=STEP_DATA_1;
				ID1_Drive := FALSE;
				TMR11(IN:=TRUE,PT:= PROCESS_DELAY);
				IF TMR11.Q THEN
					ID1_Drive := TRUE;
					TMR12(IN:=TMR11.Q,PT:= PROCESS_DELAY);
					IF TMR12.Q THEN
						
						IF ID1_INP THEN
							TMR10(IN:=FALSE);
						TMR11(IN:=FALSE);
						TMR12(IN:=FALSE);
						ID1_Drive := FALSE;
						SORTER_VAR.ACTIVE_ID:=2;
						SORTER_VAR.LASER_HOME:=TRUE;
						END_IF
					END_IF
				END_IF
			END_IF
		END_IF
	//	SORTER_VAR.I_CASE:=SORTER_VAR.I_CASE+1;
		//SORTER_VAR.I_LASER_RUNNING:=FALSE;
	2:
		IF STEP_DATA_2 = 0 THEN
			SORTER_VAR.ACTIVE_ID:=3;
		ELSE
			
			IF ID2_ALARM THEN
				Reset := TRUE;
				TMR20(IN:=TRUE,PT:= PROCESS_DELAY);
				IF TMR20.Q THEN
					Reset := FALSE;
				END_IF
			ELSE
			ID2_StepData :=STEP_DATA_2;
			TMR21(IN:=TRUE,PT:= PROCESS_DELAY);
			IF TMR21.Q THEN
				ID2_Drive := TRUE;
				TMR22(IN:=TMR21.Q,PT:= PROCESS_DELAY);
				IF TMR22.Q THEN
					
					IF ID2_INP THEN
						TMR20(IN:=FALSE);
					TMR21(IN:=FALSE);
					TMR22(IN:=FALSE);
					ID2_Drive := FALSE;
						SORTER_VAR.ACTIVE_ID:=3;
					END_IF
					END_IF
			END_IF
			END_IF
		END_IF
	3:
		IF STEP_DATA_3 = 0 THEN
			SORTER_VAR.ACTIVE_ID:=4;
		ELSE
			
		IF ID3_ALARM THEN
			Reset := TRUE;
			TMR30(IN:=START_PROCESS,PT:= PROCESS_DELAY);
			IF TMR30.Q THEN
				Reset := FALSE;
			END_IF
		ELSE
		
		ID3_StepData :=STEP_DATA_3;
		TMR31(IN:=TRUE,PT:= PROCESS_DELAY);
		IF TMR31.Q THEN
			
			ID3_DRIVE := TRUE;	
			TMR32(IN:=TMR31.Q,PT:= PROCESS_DELAY);
			
			IF TMR32.Q THEN
				
				IF ID3_INP THEN
				SORTER_VAR.ACTIVE_ID:=4;
ID3_Drive := FALSE;
				TMR30(IN:=FALSE);
				TMR31(IN:=FALSE);
				TMR32(IN:=FALSE);
				END_IF
			END_IF
		END_IF
		END_IF
	END_IF
4:
		IF STEP_DATA_4 = 0 THEN
			SORTER_VAR.ACTIVE_ID:=5;
		ELSE
			IF ID4_ALARM THEN
				Reset := TRUE;
				TMR40(IN:=TRUE,PT:= PROCESS_DELAY);
				IF TMR40.Q THEN
					Reset := FALSE;
				END_IF
			ELSE
			IF NOT ID4_READY THEN
				IF ID4_SVRE THEN
					ID4_SETUP :=TRUE;
					IF ID4_INP THEN
						ID4_READY:=TRUE;
					END_IF
				END_IF
			ELSE

			ID4_StepData :=STEP_DATA_4;
			TMR41(IN:=TRUE,PT:= PROCESS_DELAY);
			IF TMR41.Q THEN
				ID4_Drive := TRUE;
				TMR42(IN:=TMR41.Q,PT:= PROCESS_DELAY);
				
				IF TMR42.Q THEN
			
					IF ID4_INP THEN
						SORTER_VAR.ACTIVE_ID:=5;
								ID4_Drive := FALSE;
					TMR40(IN:=FALSE);
					TMR41(IN:=FALSE);
					TMR42(IN:=FALSE);
					END_IF
				END_IF
			END_IF
			END_IF
			END_IF
		END_IF
	5:
		IF STEP_DATA_5 = 0 THEN
			SORTER_VAR.ACTIVE_ID:=0;
		ELSE
			
			IF ID5_ALARM THEN
				Reset := TRUE;
				TMR50(IN:=TRUE,PT:= PROCESS_DELAY);
				IF TMR50.Q THEN
					Reset := FALSE;
				END_IF
			ELSE
				IF NOT ID5_READY THEN
				IF ID5_SVRE THEN
					ID5_SETUP :=TRUE;
					IF ID5_INP THEN
						ID5_READY:=TRUE;
					END_IF
				END_IF
			ELSE
			ID5_StepData :=STEP_DATA_5;
			TMR51(IN:=TRUE,PT:= PROCESS_DELAY);
			IF TMR51.Q THEN
				ID5_Drive := TRUE;	
				TMR52(IN:=TMR51.Q,PT:= PROCESS_DELAY);
				IF TMR52.Q THEN
					
					IF ID5_INP THEN
					SORTER_VAR.ACTIVE_ID:=0;
ID5_Drive := FALSE;
					TMR50(IN:=FALSE);
					TMR51(IN:=FALSE);
					TMR52(IN:=FALSE);
				END_IF
				END_IF
			END_IF
			END_IF
			END_IF
		END_IF
		
END_CASE 

	//START_PROCESS := FALSE;
END_IF
TMR7(IN:=reset,PT:= T#1S);
IF  tmr7.Q THEN
	reset:=FALSE;
END_IF
IF ID1_ALARM OR ID2_ALARM OR ID3_ALARM OR ID4_ALARM OR ID5_ALARM THEN
	reset:=TRUE;
	INPUT_VAR.ALARM1:=ID1_ALARM OR ID2_ALARM OR ID3_ALARM OR ID4_ALARM OR ID5_ALARM;
ELSE
	reset:=FALSE;
END_IF
IF reset THEN
	ID1_Reset := TRUE;
	ID2_Reset := TRUE;
	ID3_Reset := TRUE;
	ID4_Reset := TRUE;
	ID5_Reset := TRUE;
	TMR_ACTIVATE_RESET(IN:=TRUE,PT:=T#10S);
	IF TMR_ACTIVATE_RESET.Q THEN
		TMR_RES_CARTSN(IN:=TRUE,PT:=T#0.5S);
	END_IF
	
ELSE
	TMR_ACTIVATE_RESET(IN:=FALSE);
	TMR_RES_CARTSN(IN:=FALSE);
	ID1_Reset := FALSE;
	ID2_Reset := FALSE;
	ID3_Reset := FALSE;
	ID4_Reset := FALSE;
	ID5_Reset := FALSE;
END_IF
SORTER_VAR.O_RESET_CARTESSIAN := TMR_RES_CARTSN.Q;

END_PROGRAM

// ---- POUs/LASER/LASER_PROG.TcPOU
PROGRAM LASER_PROG
VAR
	
	PULS1: TON;
	PULS2: TON;
	CNT1: CTU;
	LOTBOX_ACC: INT;
	LOTBOX_ACC1: INT;
	LOTBOX_TEMP1: INT;
	LOTBOX_TEMP2: INT;
	LOTBOX_TEMP3: INT;
	LOTBOX_TEMP4: INT;
	NGBOX_TEMP: INT;
	NGBOX_TEMP1: INT;
	NGBOX_TEMP2: INT;
	NGBOX_TEMP3: INT;
	NGBOX_TEMP4: INT;
	NGBOX_ACC: INT;
END_VAR


PULS1(IN:=NOT PULS2.Q,PT:=T#0.5S);
PULS2(IN:=PULS1.Q,PT:=T#1S);
CNT1(CU:=PULS1.Q,RESET:=CNT1.Q,PV:=9);
(*
IF CNT1.CV=1 THEN
	SORTER_VAR.O_NG_BOX_INDICATOR_4:=TRUE;
END_IF
IF CNT1.CV=2 THEN
	SORTER_VAR.O_NG_BOX_INDICATOR_3:=TRUE;
END_IF
IF CNT1.CV=3 THEN
	SORTER_VAR.O_NG_BOX_INDICATOR_2:=TRUE;
END_IF
IF CNT1.CV=4 THEN
	SORTER_VAR.O_NG_BOX_INDICATOR_1:=TRUE;
END_IF
IF CNT1.CV=5 THEN
	SORTER_VAR.O_LOT_BOX_INDICATOR_4:=TRUE;
END_IF
IF CNT1.CV=6 THEN
	SORTER_VAR.O_LOT_BOX_INDICATOR_3:=TRUE;
END_IF
IF CNT1.CV=7 THEN
	SORTER_VAR.O_LOT_BOX_INDICATOR_2:=TRUE;
END_IF
IF CNT1.CV=8 THEN
	SORTER_VAR.O_LOT_BOX_INDICATOR_1:=TRUE;
END_IF
IF CNT1.Q THEN
	SORTER_VAR.O_LOT_BOX_INDICATOR_1:=FALSE;
	SORTER_VAR.O_LOT_BOX_INDICATOR_2:=FALSE;
	SORTER_VAR.O_LOT_BOX_INDICATOR_3:=FALSE;
	SORTER_VAR.O_LOT_BOX_INDICATOR_4:=FALSE;
	SORTER_VAR.O_NG_BOX_INDICATOR_1:=FALSE;
	SORTER_VAR.O_NG_BOX_INDICATOR_2:=FALSE;
	SORTER_VAR.O_NG_BOX_INDICATOR_3:=FALSE;
	SORTER_VAR.O_NG_BOX_INDICATOR_4:=FALSE;
END_IF
*)
IF SORTER_VAR.I_LOTBOX_DETECT_1 THEN
	SORTER_VAR.O_LOT_BOX_INDICATOR_1:=PULS1.Q;
	LOTBOX_TEMP1:=1;
ELSE
	SORTER_VAR.O_LOT_BOX_INDICATOR_1:=FALSE;
	LOTBOX_TEMP1:=0;
END_IF

IF SORTER_VAR.I_LOTBOX_DETECT_2 THEN
	SORTER_VAR.O_LOT_BOX_INDICATOR_2:=PULS1.Q;
	LOTBOX_TEMP2:=1;
	ELSE
	LOTBOX_TEMP2:=0;
	SORTER_VAR.O_LOT_BOX_INDICATOR_2:=FALSE;
END_IF

IF SORTER_VAR.I_LOTBOX_DETECT_3 THEN
	SORTER_VAR.O_LOT_BOX_INDICATOR_3:=PULS1.Q;
	LOTBOX_TEMP3:=1;
	ELSE
	SORTER_VAR.O_LOT_BOX_INDICATOR_3:=FALSE;
	LOTBOX_TEMP3:=0;
END_IF

IF SORTER_VAR.I_LOTBOX_DETECT_4 THEN
	SORTER_VAR.O_LOT_BOX_INDICATOR_4:=PULS1.Q;
	LOTBOX_TEMP4:=1;
	ELSE
	SORTER_VAR.O_LOT_BOX_INDICATOR_4:=FALSE;
	LOTBOX_TEMP4:=0;
END_IF
LOTBOX_ACC:=LOTBOX_TEMP1 +LOTBOX_TEMP2+LOTBOX_TEMP3+LOTBOX_TEMP4;

IF LOTBOX_ACC >=3 THEN
	//SORTER_VAR.O_TOWER_LAMP_BUZZER :=TRUE;
	ELSE
	SORTER_VAR.O_TOWER_LAMP_BUZZER :=FALSE;
END_IF

IF NOT SORTER_VAR.I_NG_BOX_DETECT_1 THEN
		SORTER_VAR.O_NG_BOX_INDICATOR_1:=PULS1.Q;
		NGBOX_TEMP1:=1;
		ELSE
		SORTER_VAR.O_NG_BOX_INDICATOR_1:=FALSE;
		NGBOX_TEMP1:=0;
END_IF

IF NOT SORTER_VAR.I_NG_BOX_DETECT_2 THEN
		SORTER_VAR.O_NG_BOX_INDICATOR_2:=PULS1.Q;
		NGBOX_TEMP2:=1;
		ELSE
		SORTER_VAR.O_NG_BOX_INDICATOR_2:=FALSE;
		NGBOX_TEMP2:=0;
END_IF

IF NOT SORTER_VAR.I_NG_BOX_DETECT_3 THEN
		SORTER_VAR.O_NG_BOX_INDICATOR_3:=PULS1.Q;
		NGBOX_TEMP3:=1;
		ELSE
		SORTER_VAR.O_NG_BOX_INDICATOR_3:=FALSE;
		NGBOX_TEMP3:=0;
END_IF

IF NOT SORTER_VAR.I_NG_BOX_DETECT_4 THEN
		SORTER_VAR.O_NG_BOX_INDICATOR_4:=PULS1.Q;
		NGBOX_TEMP4:=1;
		ELSE
		SORTER_VAR.O_NG_BOX_INDICATOR_4:=FALSE;
		NGBOX_TEMP4:=0;
END_IF
NGBOX_ACC:=NGBOX_TEMP1+NGBOX_TEMP2+NGBOX_TEMP3+NGBOX_TEMP4;
IF NGBOX_ACC >=3 THEN
	//SORTER_VAR.O_TOWER_LAMP_BUZZER :=TRUE;
	ELSE
	SORTER_VAR.O_TOWER_LAMP_BUZZER :=FALSE;
END_IF

END_PROGRAM

// ---- POUs/LASER/LOAD_LASER.TcPOU
PROGRAM LOAD_LASER
VAR_INPUT

END_VAR

VAR
	TMR_DELAY: TON;
	TMR1:TON;
	TMR_STOPPER_A: TON;
	TMR_STOPPER_B: TON;
	TMR_DLY: TON;
	TMR_DLY2: TON;

END_VAR

CASE SORTER_VAR.I_CASE OF
0: //standby near lotbox
	IF SORTER_VAR.ACTIVE_ID=6 THEN
		SORTER_VAR.ACTIVE_ID:=1;
	END_IF
	SORTER_VAR.TRANSPORT_IDX:=		SORTER_VAR.I_CURRENT_TRANSACTION.TRANSPORT_INDEX;
	SORTER_VAR.STATION_LOAD_IDX:=	SORTER_VAR.I_CURRENT_TRANSACTION.STATION_NUMBER_LOAD;
	SORTER_VAR.JIG_LOAD_IDX:=		SORTER_VAR.I_CURRENT_TRANSACTION.JIG_INDEX_LOAD;
	
	IF SORTER_VAR.TRANSPORT_IDX=0 AND SORTER_VAR.STATION_LOAD_IDX=0 AND SORTER_VAR.JIG_LOAD_IDX=0 THEN
		SORTER_VAR.TRANSPORT_IDX:=		SORTER_VAR.I_CURRENT_TRANSACTION.TRANSPORT_INDEX;
		SORTER_VAR.STATION_LOAD_IDX:=	SORTER_VAR.I_CURRENT_TRANSACTION.STATION_NUMBER_LOAD;
		SORTER_VAR.JIG_LOAD_IDX:=		SORTER_VAR.I_CURRENT_TRANSACTION.JIG_INDEX_LOAD;
	ELSE
		
	CASE SORTER_VAR.TRANSPORT_IDX OF
		2 : LASER_MOVE(STEP_DATA_1:=SORTER_VAR.STATION_LOAD_IDX,
				STEP_DATA_2:=0,
				STEP_DATA_3:=SORTER_VAR.JIG_LOAD_IDX,
				STEP_DATA_4:=0,
				STEP_DATA_5:=1);
				SORTER_VAR.O_STOPPER_TRANSFER_B:=FALSE;
				//SORTER_VAR.I_LOADING_DONE_B:=FALSE;
		1 : LASER_MOVE(STEP_DATA_1:=SORTER_VAR.STATION_LOAD_IDX,
				STEP_DATA_2:=0,
				STEP_DATA_3:=SORTER_VAR.JIG_LOAD_IDX,
				STEP_DATA_4:=1,
				STEP_DATA_5:=0);
				SORTER_VAR.O_STOPPER_TRANSFER_A:=FALSE;
				//SORTER_VAR.I_LOADING_DONE_A:=FALSE;
	END_CASE
END_IF			
	SORTER_VAR.O_VACUUM_On:=FALSE;
	SORTER_VAR.O_VACUUM_OFF:=FALSE;	
	SORTER_VAR.O_CARTESSIAN_GRIPPER_ON:=FALSE;
	SORTER_VAR.O_CARTESSIAN_GRIPPER_OFF:=TRUE;
	TMR_DLY(IN:=FALSE);
			
1: //standby near lotbox
	
	IF SORTER_VAR.ACTIVE_ID=6 THEN
		SORTER_VAR.ACTIVE_ID:=1;
	END_IF
	
		LASER_MOVE(STEP_DATA_1:=SORTER_VAR.STATION_LOAD_IDX,
				STEP_DATA_2:=3,
				STEP_DATA_3:=SORTER_VAR.JIG_LOAD_IDX,
				STEP_DATA_4:=0,
				STEP_DATA_5:=0);

		CASE SORTER_VAR.TRANSPORT_IDX OF
		1:
			SORTER_VAR.I_LOADING_DONE_A:=FALSE;
		
		2:
			SORTER_VAR.I_LOADING_DONE_B:=FALSE;
		END_CASE
			
2://vacuum position 
	IF SORTER_VAR.ACTIVE_ID=6 THEN
		SORTER_VAR.ACTIVE_ID:=1;
	END_IF
	SORTER_VAR.I_CASE:=SORTER_VAR.I_CASE+1;
3://vacuum position 
	IF SORTER_VAR.ACTIVE_ID=6 THEN
		SORTER_VAR.ACTIVE_ID:=1; 
	END_IF
	SORTER_VAR.I_CASE:=SORTER_VAR.I_CASE+1;

4://vacuum position 
	IF SORTER_VAR.ACTIVE_ID=6 THEN
		SORTER_VAR.ACTIVE_ID:=1;
	END_IF
	SORTER_VAR.O_VACUUM_ON:=TRUE;
	SORTER_VAR.O_VACUUM_OFF:=FALSE;

	//CHECK JIG LASER PRESENCE	
LASER_MOVE(STEP_DATA_1:=SORTER_VAR.STATION_LOAD_IDX,
				STEP_DATA_2:=4,
				STEP_DATA_3:=13,///JIG_LOAD_IDX,
				STEP_DATA_4:=0,
				STEP_DATA_5:=0);

(*		
	IF  SORTER_VAR.O_VACUUM_ON THEN
		TMR1(IN:=TRUE,PT:=T#2S);
		IF TMR1.Q THEN
			IF  SORTER_VAR.I_VACUUM_ON AND SORTER_VAR.O_VACUUM_ON THEN
				SORTER_VAR.JIG_LASER_PRESENCE :=TRUE;
				
				LASER_MOVE(STEP_DATA_1:=7,
				STEP_DATA_2:=4,
				STEP_DATA_3:=JIG_LOAD_IDX,
				STEP_DATA_4:=0,
				STEP_DATA_5:=0);
			ELSE
				SORTER_VAR.JIG_LASER_PRESENCE :=FALSE;	
				LASER_MOVE(STEP_DATA_1:=STATION_LOAD_IDX,
				STEP_DATA_2:=2,
				STEP_DATA_3:=JIG_LOAD_IDX,
				STEP_DATA_4:=0,
				STEP_DATA_5:=0);
				
				LASER_MOVE(STEP_DATA_1:=STATION_LOAD_IDX,
				STEP_DATA_2:=1,
				STEP_DATA_3:=JIG_LOAD_IDX,
				STEP_DATA_4:=0,
				STEP_DATA_5:=0);
				
				TMR_DELAY(IN:=TRUE,PT:=T#2S);
				IF TMR_DELAY.Q THEN
					FLAG_VAR.ALLOW_EXECUTE_LOAD_LASER:=FALSE;
					JIG_LOAD_IDX:=JIG_LOAD_IDX+0;
					SORTER_VAR.I_CASE:=0;
					TMR1(IN:=FALSE);
					SORTER_VAR.O_VACUUM_ON:=FALSE;
					SORTER_VAR.O_VACUUM_OFF:=FALSE;
				END_IF
			END_IF
		END_IF 
	END_IF
*)
				

5://vacuum position 
	IF SORTER_VAR.ACTIVE_ID=6 THEN
		SORTER_VAR.ACTIVE_ID:=1;
	END_IF
	SORTER_VAR.O_CARTESSIAN_GRIPPER_ON:=TRUE;
	SORTER_VAR.O_CARTESSIAN_GRIPPER_OFF:=FALSE;
	TMR_DLY2(IN:=TRUE,PT:=T#2S);
	IF TMR_DLY2.Q THEN
		
		IF SORTER_VAR.I_CARTESSIAN_GRIPPER_ON THEN
			LASER_MOVE(STEP_DATA_1:=SORTER_VAR.STATION_LOAD_IDX,//9,
				STEP_DATA_2:=2,
				STEP_DATA_3:=9,//JIG_LOAD_IDX,
				STEP_DATA_4:=0,
				STEP_DATA_5:=0);
			TMR_DLY(IN:=FALSE);
		ELSE
			TMR_DLY(IN:=TRUE,PT:=T#3S);
			IF TMR_DLY.Q THEN
				SORTER_VAR.I_CASE:=50;
				TMR_DLY(IN:=FALSE);
			END_IF
		END_IF
	END_IF	

6://gripping position
	IF SORTER_VAR.ACTIVE_ID=6 THEN
		SORTER_VAR.ACTIVE_ID:=1;
	END_IF

	LASER_MOVE(STEP_DATA_1:=SORTER_VAR.TRANSPORT_IDX+5,
				STEP_DATA_2:=2,
				STEP_DATA_3:=12,
				STEP_DATA_4:=0,
				STEP_DATA_5:=0);


7://placing onto LASER transport
	IF SORTER_VAR.ACTIVE_ID=6 THEN
		SORTER_VAR.ACTIVE_ID:=1;
	END_IF
	LASER_MOVE(STEP_DATA_1:=SORTER_VAR.TRANSPORT_IDX+5,
				STEP_DATA_2:=6,
				STEP_DATA_3:=11,
				STEP_DATA_4:=0,
				STEP_DATA_5:=0);
	
8://homing
	IF SORTER_VAR.ACTIVE_ID=6 THEN
		SORTER_VAR.ACTIVE_ID:=1;
	END_IF
	SORTER_VAR.O_CARTESSIAN_GRIPPER_ON:=FALSE;
	SORTER_VAR.O_CARTESSIAN_GRIPPER_OFF:=TRUE;
	IF SORTER_VAR.I_CARTESSIAN_GRIPPER_OFF THEN
		LASER_MOVE(STEP_DATA_1:=SORTER_VAR.TRANSPORT_IDX+5,
				STEP_DATA_2:=0,
				STEP_DATA_3:=18,
				STEP_DATA_4:=0,
				STEP_DATA_5:=0);
	END_IF			
9://homing
	IF SORTER_VAR.ACTIVE_ID=6 THEN
		SORTER_VAR.ACTIVE_ID:=1;
	END_IF
	LASER_MOVE(STEP_DATA_1:=SORTER_VAR.TRANSPORT_IDX+5,
				STEP_DATA_2:=1,
				STEP_DATA_3:=10,
				STEP_DATA_4:=0,
				STEP_DATA_5:=0);
	
10://pusH LASER transport
	IF SORTER_VAR.ACTIVE_ID=6 THEN
		SORTER_VAR.ACTIVE_ID:=1;
	END_IF
	SORTER_VAR.O_VACUUM_OFF:=FALSE;

	CASE SORTER_VAR.TRANSPORT_IDX OF
		2 :
			//IF  SORTER_VAR.I_LASER_TRANSFER_AT_FRONT_B THEN
				LASER_MOVE(STEP_DATA_1:=0,
				STEP_DATA_2:=0,
				STEP_DATA_3:=0,
				STEP_DATA_4:=0,
				STEP_DATA_5:=2);
			//END_IF
				 
		1 : 
			//IF  SORTER_VAR.I_LASER_TRANSFER_AT_FRONT_A THEN
				LASER_MOVE(STEP_DATA_1:=0,
				STEP_DATA_2:=0,
				STEP_DATA_3:=0,
				STEP_DATA_4:=2,
				STEP_DATA_5:=0);
			//END_IF
	END_CASE	

11:
		TMR_DLY(IN:=FALSE);
		SORTER_VAR.O_NG_BUFFER_ON:=FALSE;
		SORTER_VAR.O_NG_BUFFER_OFF:=FALSE;
		CASE SORTER_VAR.TRANSPORT_IDX OF
		1:	
			IF SORTER_VAR.I_LASER_TRANSFER_AT_FRONT_A THEN
				TMR_STOPPER_A(IN:=TRUE,PT:=T#1S);
				IF TMR_STOPPER_A.Q THEN
					SORTER_VAR.O_STOPPER_TRANSFER_A:=TRUE;
					SORTER_VAR.I_LOADING_DONE_A:=TRUE;
					TMR1(IN:=FALSE);
					TMR_DELAY(IN:=FALSE);
					FLAG_VAR.ALLOW_EXECUTE_LOAD_LASER:=FALSE;	
					SORTER_VAR.I_CASE:=100;
					SORTER_VAR.O_VACUUM_On:=FALSE;
					SORTER_VAR.O_VACUUM_OFF:=FALSE;
				END_IF
			END_IF
	
			2:
			IF SORTER_VAR.I_LASER_TRANSFER_AT_FRONT_B THEN
				
				TMR_STOPPER_B(IN:=TRUE,PT:=T#1S);
				IF TMR_STOPPER_B.Q THEN
					SORTER_VAR.O_STOPPER_TRANSFER_B:=TRUE;	
					SORTER_VAR.I_LOADING_DONE_B:=TRUE;
					TMR1(IN:=FALSE);
					TMR_DELAY(IN:=FALSE);
					FLAG_VAR.ALLOW_EXECUTE_LOAD_LASER:=FALSE;	
					SORTER_VAR.I_CASE:=100;
					SORTER_VAR.O_VACUUM_On:=FALSE;
					SORTER_VAR.O_VACUUM_OFF:=FALSE;
				END_IF
			END_IF
	END_CASE
	
50:
LASER_MOVE(STEP_DATA_1:=0,
				STEP_DATA_2:=0,
				STEP_DATA_3:=0,
				STEP_DATA_4:=0,
				STEP_DATA_5:=0);
		
51:
	FLAG_VAR.ALLOW_EXECUTE_LOAD_LASER:=FALSE;
	SORTER_VAR.I_CASE:=100;
100:
	SORTER_VAR.O_VACUUM_On:=FALSE;
	SORTER_VAR.O_VACUUM_OFF:=FALSE;
	TMR1(IN:=FALSE);
	TMR_DELAY(IN:=FALSE);
	FLAG_VAR.ALLOW_EXECUTE_LOAD_LASER:=FALSE;								
								
END_CASE 
(*ELSE
	LASER_MOVE(STEP_DATA_1:=0,
				STEP_DATA_2:=0,
				STEP_DATA_3:=0,
				STEP_DATA_4:=0,
				STEP_DATA_5:=0);
END_IF*)

END_PROGRAM

// ---- POUs/LASER/LOAD_NG.TcPOU
PROGRAM LOAD_NG
VAR
	DELAY: TON;

	TMR_DLY: TON;
END_VAR

IF NOT SORTER_VAR.I_NG_HOME THEN
	SORTER_VAR.O_NG_DATA_OUTPUT1:=TRUE;
	SORTER_VAR.O_NG_DATA_OUTPUT2:=TRUE;
	SORTER_VAR.O_NG_DATA_OUTPUT3:=TRUE;
	SORTER_VAR.O_NG_DATA_OUTPUT4:=TRUE;
	TMR_DLY(IN:=TRUE,PT:=T#1S);
	IF TMR_DLY.Q THEN
		SORTER_VAR.O_NG_DATA_OUTPUT1:=FALSE;
		SORTER_VAR.O_NG_DATA_OUTPUT2:=FALSE;
		SORTER_VAR.O_NG_DATA_OUTPUT3:=FALSE;
		SORTER_VAR.O_NG_DATA_OUTPUT4:=FALSE;
		SORTER_VAR.I_NG_HOME:=TRUE;
		TMR_DLY(IN:=FALSE);
	END_IF
ELSE
CASE SORTER_VAR.I_NG_CASE OF
	1:	IF SORTER_VAR.ACTIVE_ID=6 THEN
			SORTER_VAR.ACTIVE_ID:=1;
		END_IF
		SORTER_VAR.LOAD_NG_IDX :=SORTER_VAR.I_CURRENT_TRANSACTION.JIG_INDEX_LOAD_NG;
		
		SORTER_VAR.O_NG_DATA_OUTPUT1:=TRUE;
		SORTER_VAR.O_NG_DATA_OUTPUT2:=FALSE;
		SORTER_VAR.O_NG_DATA_OUTPUT3:=FALSE;
		SORTER_VAR.O_NG_DATA_OUTPUT4:=FALSE;
		
		SORTER_VAR.I_LOADING_DONE_NG:=FALSE;
		SORTER_VAR.O_CARTESSIAN_GRIPPER_ON:=FALSE;
		SORTER_VAR.O_CARTESSIAN_GRIPPER_OFF:=TRUE;
//HOMING POSITION	
		LASER_MOVE(STEP_DATA_1:=0,
				STEP_DATA_2:=0,
				STEP_DATA_3:=21,
				STEP_DATA_4:=0,
				STEP_DATA_5:=0);
				
	2:	IF SORTER_VAR.ACTIVE_ID=6 THEN
			SORTER_VAR.ACTIVE_ID:=1;
		END_IF
//NEAR BOX POSITION	
		LASER_MOVE(STEP_DATA_1:=5,
				STEP_DATA_2:=3,
				STEP_DATA_3:=SORTER_VAR.LOAD_NG_IDX+19,
				STEP_DATA_4:=0,
				STEP_DATA_5:=0);
				
	3:	IF SORTER_VAR.ACTIVE_ID=6 THEN
			SORTER_VAR.ACTIVE_ID:=1;
		END_IF
//ON BOX POSITION	
		LASER_MOVE(STEP_DATA_1:=5,
				STEP_DATA_2:=8,
				STEP_DATA_3:=SORTER_VAR.LOAD_NG_IDX+19,
				STEP_DATA_4:=0,
				STEP_DATA_5:=0);

	4:	IF SORTER_VAR.ACTIVE_ID=6 THEN
			SORTER_VAR.ACTIVE_ID:=1;
		END_IF
			SORTER_VAR.O_CARTESSIAN_GRIPPER_ON:=TRUE;
			SORTER_VAR.O_CARTESSIAN_GRIPPER_OFF:=FALSE;
			IF SORTER_VAR.I_CARTESSIAN_GRIPPER_ON THEN
//GRIP ON AND LIFT
				LASER_MOVE(STEP_DATA_1:=5,
				STEP_DATA_2:=8,
				STEP_DATA_3:=14,
				STEP_DATA_4:=0,
				STEP_DATA_5:=0);				
			END_IF
	5:	IF SORTER_VAR.ACTIVE_ID=6 THEN
			SORTER_VAR.ACTIVE_ID:=1;
		END_IF
//MOVE BACK	
		LASER_MOVE(STEP_DATA_1:=5,//SORTER_VAR.I_CURRENT_TRANSACTION.TRANSPORT_INDEX+5,
				STEP_DATA_2:=2,
				STEP_DATA_3:=10,//SORTER_VAR.I_CURRENT_TRANSACTION.JIG_INDEX_LOAD_NG,
				STEP_DATA_4:=0,
				STEP_DATA_5:=0);
				
	6:	IF SORTER_VAR.ACTIVE_ID=6 THEN
			SORTER_VAR.ACTIVE_ID:=1;
		END_IF
//ABOVE TRANSFER POSITION
		LASER_MOVE(STEP_DATA_1:=8,
				STEP_DATA_2:=0,
				STEP_DATA_3:=12,
				STEP_DATA_4:=0,
				STEP_DATA_5:=0);

	7:	IF SORTER_VAR.ACTIVE_ID=6 THEN
			SORTER_VAR.ACTIVE_ID:=1;
		END_IF
//ON TRANSFER POSITION
		LASER_MOVE(STEP_DATA_1:=8,
				STEP_DATA_2:=0,
				STEP_DATA_3:=11,
				STEP_DATA_4:=0,
				STEP_DATA_5:=0);	
				
	8:	IF SORTER_VAR.ACTIVE_ID=6 THEN
			SORTER_VAR.ACTIVE_ID:=1;
		END_IF
		SORTER_VAR.O_CARTESSIAN_GRIPPER_ON:=FALSE;
		SORTER_VAR.O_CARTESSIAN_GRIPPER_OFF:=TRUE;
		IF SORTER_VAR.I_CARTESSIAN_GRIPPER_OFF THEN
//GRIP OFF AND MOVE BACK
		LASER_MOVE(STEP_DATA_1:=8,
				STEP_DATA_2:=1,
				STEP_DATA_3:=11,
				STEP_DATA_4:=0,
				STEP_DATA_5:=0);	
		END_IF
	9:	IF SORTER_VAR.ACTIVE_ID=6 THEN
			SORTER_VAR.ACTIVE_ID:=1;
		END_IF
//HOME POSITION
		LASER_MOVE(STEP_DATA_1:=0,
				STEP_DATA_2:=0,
				STEP_DATA_3:=12,
				STEP_DATA_4:=0,
				STEP_DATA_5:=0);
	10:
		SORTER_VAR.O_NG_DATA_OUTPUT1:=FALSE;
		SORTER_VAR.O_NG_DATA_OUTPUT2:=TRUE;
		SORTER_VAR.O_NG_DATA_OUTPUT3:=FALSE;
		SORTER_VAR.O_NG_DATA_OUTPUT4:=FALSE;
		IF SORTER_VAR.I_NG_TRANSFER_AT_FRONT THEN
			SORTER_VAR.I_LOADING_DONE_NG:=TRUE;
			SORTER_VAR.O_NG_DATA_OUTPUT2:=FALSE;
			SORTER_VAR.I_NG_CASE:=100;
			FLAG_VAR.ALLOW_EXECUTE_LOAD_NG:=FALSE;
		END_IF
		
	100: 	FLAG_VAR.ALLOW_EXECUTE_LOAD_NG:=FALSE;
			SORTER_VAR.O_CARTESSIAN_GRIPPER_ON:=FALSE;
			SORTER_VAR.O_CARTESSIAN_GRIPPER_OFF:=FALSE;
			
END_CASE
END_IF

END_PROGRAM

// ---- POUs/LASER/RETURN_LASER.TcPOU
PROGRAM RETURN_LASER
VAR_INPUT

END_VAR

VAR
	TMR_DELAY: TON;
	TMR_DELAY1: TON;
	TMR_DELAY2: TON;
END_VAR


IF SORTER_VAR.TRANSPORT_IDX=0 AND SORTER_VAR.STATION_RETURN_IDX=0 AND SORTER_VAR.JIG_RETURN_IDX=0 THEN
	SORTER_VAR.TRANSPORT_IDX:=SORTER_VAR.I_CURRENT_TRANSACTION.TRANSPORT_INDEX;
	SORTER_VAR.STATION_RETURN_IDX:=SORTER_VAR.I_CURRENT_TRANSACTION.STATION_NUMBER_LOAD;
	SORTER_VAR.JIG_RETURN_IDX:=SORTER_VAR.I_CURRENT_TRANSACTION.JIG_INDEX_LOAD;
ELSE
CASE SORTER_VAR.I_CASE OF
0: //standby near lotbox
	IF SORTER_VAR.ACTIVE_ID=6 THEN
		SORTER_VAR.ACTIVE_ID:=1;
	END_IF
	SORTER_VAR.TRANSPORT_IDX:=SORTER_VAR.I_CURRENT_TRANSACTION.TRANSPORT_INDEX;
	SORTER_VAR.STATION_RETURN_IDX:=SORTER_VAR.I_CURRENT_TRANSACTION.STATION_NUMBER_RETURN;
	SORTER_VAR.JIG_RETURN_IDX:=SORTER_VAR.I_CURRENT_TRANSACTION.JIG_INDEX_RETURN;
	CASE SORTER_VAR.I_CURRENT_TRANSACTION.TRANSPORT_INDEX OF
		2 : 
			SORTER_VAR.O_STOPPER_TRANSFER_B:=FALSE;			
			LASER_MOVE(STEP_DATA_1:=0,//3,
				STEP_DATA_2:=0,
				STEP_DATA_3:=12,
				STEP_DATA_4:=0,
				STEP_DATA_5:=1);
				SORTER_VAR.I_RETURN_DONE_B:=FALSE;
		1 : 
			SORTER_VAR.O_STOPPER_TRANSFER_A:=FALSE;
			LASER_MOVE(STEP_DATA_1:=0,//3,
				STEP_DATA_2:=0,
				STEP_DATA_3:=12,
				STEP_DATA_4:=1,
				STEP_DATA_5:=0);
				SORTER_VAR.I_RETURN_DONE_A:=FALSE;
	END_CASE			
	SORTER_VAR.O_VACUUM_On:=FALSE;
	SORTER_VAR.O_VACUUM_OFF:=FALSE;	
	TMR_DELAY(IN:=FALSE);
	SORTER_VAR.O_CARTESSIAN_GRIPPER_ON:=FALSE;
	SORTER_VAR.O_CARTESSIAN_GRIPPER_OFF:=TRUE;

1://ready for picking up
	IF SORTER_VAR.ACTIVE_ID=6 THEN
		SORTER_VAR.ACTIVE_ID:=1;
	END_IF
	SORTER_VAR.O_NG_BUFFER_ON:=TRUE;
	SORTER_VAR.O_NG_BUFFER_OFF:=FALSE;
	CASE SORTER_VAR.TRANSPORT_IDX OF
	1:
		SORTER_VAR.I_RETURN_DONE_A:=FALSE;
		IF NOT SORTER_VAR.I_LASER_TRANSFER_AT_BACK_A THEN
			SORTER_VAR.I_CASE:=0;
		ELSE
			LASER_MOVE(STEP_DATA_1:=0,
				STEP_DATA_2:=1,
				STEP_DATA_3:=11,
				STEP_DATA_4:=1,
				STEP_DATA_5:=0);	
		END_IF
	2:
		SORTER_VAR.I_RETURN_DONE_B:=FALSE;
		IF NOT SORTER_VAR.I_LASER_TRANSFER_AT_BACK_B THEN
			SORTER_VAR.I_CASE:=0;
		ELSE
			LASER_MOVE(STEP_DATA_1:=0,
				STEP_DATA_2:=1,
				STEP_DATA_3:=11,
				STEP_DATA_4:=0,
				STEP_DATA_5:=1);	
		END_IF
	END_CASE
2://ready for picking up
	IF SORTER_VAR.ACTIVE_ID=6 THEN
		SORTER_VAR.ACTIVE_ID:=1;
	END_IF

	CASE SORTER_VAR.TRANSPORT_IDX OF
	1:		
				
//IF SORTER_VAR.I_LASER_TRANSFER_AT_BACK_A THEN
		LASER_MOVE(STEP_DATA_1:=SORTER_VAR.TRANSPORT_IDX+5,
				STEP_DATA_2:=1,
				STEP_DATA_3:=18,
				STEP_DATA_4:=0,
				STEP_DATA_5:=0);
		//END_IF
	2:
		//IF SORTER_VAR.I_LASER_TRANSFER_AT_BACK_B THEN
		//IF  NOT SORTER_VAR.I_LASER_TRANSFER_AT_BACK_B THEN
		LASER_MOVE(STEP_DATA_1:=SORTER_VAR.TRANSPORT_IDX+5,
				STEP_DATA_2:=1,
				STEP_DATA_3:=18,
				STEP_DATA_4:=0,
				STEP_DATA_5:=0);
		//END_IF
	END_CASE

		
3://VACUUM AND TAKEUP
	IF SORTER_VAR.ACTIVE_ID=6 THEN
		SORTER_VAR.ACTIVE_ID:=1;
	END_IF

			LASER_MOVE(STEP_DATA_1:=SORTER_VAR.TRANSPORT_IDX+5,
				STEP_DATA_2:=2,
				STEP_DATA_3:=11,
				STEP_DATA_4:=0,
				STEP_DATA_5:=0);
	
	SORTER_VAR.O_VACUUM_On:=TRUE;
	SORTER_VAR.O_VACUUM_OFF:=FALSE;
	
4://VACUUM AND TAKEUP
	IF SORTER_VAR.ACTIVE_ID=6 THEN
		SORTER_VAR.ACTIVE_ID:=1;
	END_IF

	LASER_MOVE(STEP_DATA_1:=SORTER_VAR.TRANSPORT_IDX+5,
				STEP_DATA_2:=9,
				STEP_DATA_3:=11,
				STEP_DATA_4:=0,
				STEP_DATA_5:=0);
	SORTER_VAR.O_VACUUM_On:=TRUE;
	SORTER_VAR.O_VACUUM_OFF:=FALSE;
	
5://MOVE BACK 10MM
	IF SORTER_VAR.ACTIVE_ID=6 THEN
		SORTER_VAR.ACTIVE_ID:=1;
	END_IF
	SORTER_VAR.O_CARTESSIAN_GRIPPER_ON:=TRUE;
	SORTER_VAR.O_CARTESSIAN_GRIPPER_OFF:=FALSE;
	IF SORTER_VAR.I_CARTESSIAN_GRIPPER_ON THEN
	LASER_MOVE(STEP_DATA_1:=SORTER_VAR.TRANSPORT_IDX+5,
				STEP_DATA_2:=10,
				STEP_DATA_3:=SORTER_VAR.JIG_RETURN_IDX,//12,
				STEP_DATA_4:=0,
				STEP_DATA_5:=0);
END_IF
		
6://vacuum position 
	IF SORTER_VAR.ACTIVE_ID=6 THEN
		SORTER_VAR.ACTIVE_ID:=1;
	END_IF
	//SORTER_VAR.I_CASE:=SORTER_VAR.I_CASE+1;
	
	TMR_DELAY(IN:=TRUE,PT:=T#1S);
	IF TMR_DELAY.Q THEN
			LASER_MOVE(STEP_DATA_1:=SORTER_VAR.STATION_RETURN_IDX,
				STEP_DATA_2:=3,
				STEP_DATA_3:=14,
				STEP_DATA_4:=0,
				STEP_DATA_5:=0);
	END_IF
				
7://INSERT INTO LOTBOX
	IF SORTER_VAR.ACTIVE_ID=6 THEN
		SORTER_VAR.ACTIVE_ID:=1;
	END_IF
	TMR_DELAY(IN:=FALSE);
	LASER_MOVE(STEP_DATA_1:=SORTER_VAR.STATION_RETURN_IDX,
				STEP_DATA_2:=4,
				STEP_DATA_3:=SORTER_VAR.JIG_RETURN_IDX,//16,
				STEP_DATA_4:=0,
				STEP_DATA_5:=0);
				
8://MOVE BACK
	IF SORTER_VAR.ACTIVE_ID=6 THEN
		SORTER_VAR.ACTIVE_ID:=1;
	END_IF
	TMR_DELAY2 (IN:=TRUE,PT:=T#2S);
	//IF TMR_DELAY2.Q THEN
	SORTER_VAR.O_CARTESSIAN_GRIPPER_ON:=FALSE;
	SORTER_VAR.O_CARTESSIAN_GRIPPER_OFF:=TRUE;
	IF SORTER_VAR.I_CARTESSIAN_GRIPPER_OFF THEN
		LASER_MOVE(STEP_DATA_1:=SORTER_VAR.STATION_RETURN_IDX,
				STEP_DATA_2:=10,
				STEP_DATA_3:=18,//SORTER_VAR.I_CURRENT_TRANSACTION.JIG_INDEX_RETURN,
				STEP_DATA_4:=0,
				STEP_DATA_5:=0);
	END_IF
	SORTER_VAR.O_VACUUM_On:=FALSE;
	SORTER_VAR.O_VACUUM_OFF:=TRUE;
9: //standby near lotbox
	
	IF SORTER_VAR.ACTIVE_ID=6 THEN
		SORTER_VAR.ACTIVE_ID:=1;
	END_IF
	//SORTER_VAR.I_CASE:=SORTER_VAR.I_CASE+1;
	LASER_MOVE(STEP_DATA_1:=SORTER_VAR.STATION_RETURN_IDX,
				STEP_DATA_2:=1,
				STEP_DATA_3:=10,//SORTER_VAR.I_CURRENT_TRANSACTION.JIG_INDEX_RETURN,
				STEP_DATA_4:=0,
				STEP_DATA_5:=0);

				
10://vacuum position 
	IF SORTER_VAR.ACTIVE_ID=6 THEN
		SORTER_VAR.ACTIVE_ID:=1;
	END_IF
	LASER_MOVE(STEP_DATA_1:=0,
				STEP_DATA_2:=1,
				STEP_DATA_3:=4,
				STEP_DATA_4:=0,
				STEP_DATA_5:=0);
	IF SORTER_VAR.ACTIVE_ID=3 THEN
		SORTER_VAR.O_VACUUM_ON:=FALSE;
		SORTER_VAR.O_VACUUM_OFF:=FALSE;	
	END_IF
		
100:
	SORTER_VAR.O_NG_BUFFER_ON:=FALSE;
	SORTER_VAR.O_NG_BUFFER_OFF:=FALSE;
	SORTER_VAR.O_VACUUM_On:=FALSE;
	SORTER_VAR.O_VACUUM_OFF:=FALSE;
END_CASE 
END_IF
IF SORTER_VAR.I_CASE=11 THEN
			CASE SORTER_VAR.TRANSPORT_IDX OF
		1:
			SORTER_VAR.I_RETURN_DONE_A:=TRUE;
		
		2:
			SORTER_VAR.I_RETURN_DONE_B:=TRUE;
	END_CASE
	IF SORTER_VAR.I_RETURN_DONE_A OR SORTER_VAR.I_RETURN_DONE_B THEN
		FLAG_VAR.ALLOW_EXECUTE_RETURN_LASER:=FALSE;
		TMR_DELAY(IN:=FALSE);
		TMR_DELAY1(IN:=FALSE);
		TMR_DELAY2(IN:=FALSE);
		
		SORTER_VAR.I_CASE:=100;
	END_IF
END_IF

END_PROGRAM

// ---- POUs/LASER/RETURN_NG.TcPOU
PROGRAM RETURN_NG
VAR
	DELAY: TON;
	TMR_DLY: TON;
END_VAR

 IF NOT SORTER_VAR.I_NG_HOME THEN
	SORTER_VAR.O_NG_DATA_OUTPUT1:=TRUE;
	SORTER_VAR.O_NG_DATA_OUTPUT2:=TRUE;
	SORTER_VAR.O_NG_DATA_OUTPUT3:=TRUE;
	SORTER_VAR.O_NG_DATA_OUTPUT4:=TRUE;
	TMR_DLY(IN:=TRUE,PT:=T#1S);
	IF TMR_DLY.Q THEN
		SORTER_VAR.O_NG_DATA_OUTPUT1:=FALSE;
		SORTER_VAR.O_NG_DATA_OUTPUT2:=FALSE;
		SORTER_VAR.O_NG_DATA_OUTPUT3:=FALSE;
		SORTER_VAR.O_NG_DATA_OUTPUT4:=FALSE;
		SORTER_VAR.I_NG_HOME:=TRUE;
		TMR_DLY(IN:=FALSE);
	END_IF
ELSE

CASE SORTER_VAR.I_NG_CASE OF
	1:	IF SORTER_VAR.ACTIVE_ID=6 THEN
			SORTER_VAR.ACTIVE_ID:=1;
		END_IF
		SORTER_VAR.RETURN_NG_IDX:=SORTER_VAR.I_CURRENT_TRANSACTION.JIG_INDEX_RETURN_NG;
		IF SORTER_VAR.I_NG_BUFFER_ON THEN 
		SORTER_VAR.O_NG_BUFFER_ON:=FALSE;
		SORTER_VAR.O_NG_BUFFER_OFF:=TRUE;
		END_IF
		IF SORTER_VAR.I_NG_BUFFER_OFF THEN
			SORTER_VAR.O_NG_DATA_OUTPUT1:=TRUE;
			SORTER_VAR.O_NG_DATA_OUTPUT2:=FALSE;
			SORTER_VAR.O_NG_DATA_OUTPUT3:=FALSE;
			SORTER_VAR.O_NG_DATA_OUTPUT4:=FALSE;
		END_IF
		SORTER_VAR.O_CARTESSIAN_GRIPPER_ON:=FALSE;
		SORTER_VAR.O_CARTESSIAN_GRIPPER_OFF:=TRUE;
		IF SORTER_VAR.I_NG_TRANSFER_AT_BACK THEN
			SORTER_VAR.O_NG_BUFFER_ON:=TRUE;
			SORTER_VAR.O_NG_BUFFER_OFF:=FALSE;
//HOMING POSITION	
		LASER_MOVE(STEP_DATA_1:=0,
				STEP_DATA_2:=1,
				STEP_DATA_3:=12,
				STEP_DATA_4:=0,
				STEP_DATA_5:=0);
		END_IF		
	2:	IF SORTER_VAR.ACTIVE_ID=6 THEN
			SORTER_VAR.ACTIVE_ID:=1;
		END_IF
		SORTER_VAR.O_NG_BUFFER_ON:=TRUE;
		SORTER_VAR.O_NG_BUFFER_OFF:=FALSE;
//ON TRANSFER POSITION
		LASER_MOVE(STEP_DATA_1:=0,
				STEP_DATA_2:=1,
				STEP_DATA_3:=11,
				STEP_DATA_4:=0,
				STEP_DATA_5:=0);
	
	3:	IF SORTER_VAR.ACTIVE_ID=6 THEN
			SORTER_VAR.ACTIVE_ID:=1;
		END_IF
//ON TRANSFER POSITION
		LASER_MOVE(STEP_DATA_1:=8,
				STEP_DATA_2:=2,
				STEP_DATA_3:=11,
				STEP_DATA_4:=0,
				STEP_DATA_5:=0);
		
	4:	IF SORTER_VAR.ACTIVE_ID=6 THEN
			SORTER_VAR.ACTIVE_ID:=1;
		END_IF
		SORTER_VAR.O_CARTESSIAN_GRIPPER_ON:=TRUE;
		SORTER_VAR.O_CARTESSIAN_GRIPPER_OFF:=FALSE;
		IF SORTER_VAR.I_CARTESSIAN_GRIPPER_ON THEN
//ABOVE TRANSFER POSITION
		LASER_MOVE(STEP_DATA_1:=8,
				STEP_DATA_2:=2,
				STEP_DATA_3:=SORTER_VAR.RETURN_NG_IDX+19,
				STEP_DATA_4:=0,
				STEP_DATA_5:=0);	
		END_IF
	
	5:	IF SORTER_VAR.ACTIVE_ID=6 THEN
			SORTER_VAR.ACTIVE_ID:=1;
		END_IF
//MOVE RIGHT	
		LASER_MOVE(STEP_DATA_1:=5,//SORTER_VAR.I_CURRENT_TRANSACTION.TRANSPORT_INDEX+5,
				STEP_DATA_2:=2,
				STEP_DATA_3:=14,
				STEP_DATA_4:=0,
				STEP_DATA_5:=0);
			
	6:	IF SORTER_VAR.ACTIVE_ID=6 THEN
			SORTER_VAR.ACTIVE_ID:=1;
		END_IF
//ON BOX POSITION	
		LASER_MOVE(STEP_DATA_1:=5,
				STEP_DATA_2:=8,
				STEP_DATA_3:=10,
				STEP_DATA_4:=0,
				STEP_DATA_5:=0);
	7:	IF SORTER_VAR.ACTIVE_ID=6 THEN
			SORTER_VAR.ACTIVE_ID:=1;
		END_IF
//ON BOX POSITION	AND MOVE DOWN
		LASER_MOVE(STEP_DATA_1:=5,
				STEP_DATA_2:=8,
				STEP_DATA_3:=SORTER_VAR.RETURN_NG_IDX+19,
				STEP_DATA_4:=0,
				STEP_DATA_5:=0);				
				
	8:	IF SORTER_VAR.ACTIVE_ID=6 THEN
			SORTER_VAR.ACTIVE_ID:=1;
		END_IF
		SORTER_VAR.O_CARTESSIAN_GRIPPER_ON:=FALSE;
		SORTER_VAR.O_CARTESSIAN_GRIPPER_OFF:=TRUE;
		IF SORTER_VAR.I_CARTESSIAN_GRIPPER_OFF THEN
//GRIP OFF AND MOVE BACK
				LASER_MOVE(STEP_DATA_1:=5,
				STEP_DATA_2:=1,
				STEP_DATA_3:=SORTER_VAR.RETURN_NG_IDX+19,
				STEP_DATA_4:=0,
				STEP_DATA_5:=0);				
		END_IF
	
	9:	IF SORTER_VAR.ACTIVE_ID=6 THEN
			SORTER_VAR.ACTIVE_ID:=1;
		END_IF
//HOME POSITION
		LASER_MOVE(STEP_DATA_1:=0,
				STEP_DATA_2:=0,
				STEP_DATA_3:=12,
				STEP_DATA_4:=0,
				STEP_DATA_5:=0);
	10:
		SORTER_VAR.O_NG_DATA_OUTPUT1:=FALSE;
		SORTER_VAR.O_NG_DATA_OUTPUT2:=FALSE;
		SORTER_VAR.O_NG_DATA_OUTPUT3:=FALSE;
		SORTER_VAR.O_NG_DATA_OUTPUT4:=FALSE;
		
		SORTER_VAR.I_RETURN_DONE_NG:=TRUE;
		SORTER_VAR.O_CARTESSIAN_GRIPPER_ON:=FALSE;
		SORTER_VAR.O_CARTESSIAN_GRIPPER_OFF:=FALSE;
		//IF SORTER_VAR.I_NG_TRANSFER_AT_BACK THEN
			SORTER_VAR.O_NG_DATA_OUTPUT2:=FALSE;
			SORTER_VAR.I_NG_CASE:=100;
			FLAG_VAR.ALLOW_EXECUTE_RETURN_NG:=FALSE;
		//END_IF
		
	100: 	FLAG_VAR.ALLOW_EXECUTE_RETURN_NG:=FALSE;
			SORTER_VAR.O_NG_BUFFER_ON:=FALSE;
			SORTER_VAR.O_NG_BUFFER_OFF:=FALSE;
			
END_CASE
END_IF

END_PROGRAM

// ---- POUs/LOADER/INDEXING.TcPOU
PROGRAM INDEXING
VAR
	bStartInput : BOOL;
	bServoOn : BOOL;
	bProgram0_On : BOOL;
	bProgram1_On : BOOL :=TRUE;
	bProgram2_On : BOOL :=FALSE;
	bProgram3_On : BOOL:=FALSE;
	bProgram4_On : BOOL:=FALSE;	
	bHomePositionReturn : BOOL;
	bResetInput : BOOL;
	bEmergencyInput : BOOL := TRUE;
	
	IN_POSITION_INPUT: BOOL;
	IN_POSITIONING_COMPLETION: BOOL;
	IN_START_INPUT_WAIT: BOOL;
	IN_ALARM1: BOOL;
	IN_ALARM2: BOOL;
	IN_READY_STATE: BOOL;
	T1: TON;
	TMR1: TON;
	TMR2: TON;
	TMR3: TON;
	TMR4: TON;
	TMR5: TON;
	TMR6: TON;
	TMR7: TON;
	IN_SERVO_STATUS: BOOL;
	bFirstDigit: BOOL;
	CNT1: CTU;
	ResetCount: BOOL;
	IPC: TP;
	IN_POSITIONING_COMPLET: BOOL;
	CNT2: CTU;
	START_STRAIGTHEN: BOOL;

	START_STRAIGHTEN: R_TRIG;
	START_ROTATING: R_TRIG;
	START_ROTATION: TP;
	SS: R_TRIG;
	CNT_START: CTU;
	TMR_PROCESS: TOF;
	TMR8: TON;
	TMR_OFF: TON;
	TMR_RELEASE: TON;
	INPOS: R_TRIG;
	A: BOOL;
END_VAR

INDEXING_1_VAR.DataByteOutput[0].0 := bProgram0_On;
INDEXING_1_VAR.DataByteOutput[0].1 := bProgram1_On;
INDEXING_1_VAR.DataByteOutput[0].2 := bProgram2_On;
INDEXING_1_VAR.DataByteOutput[0].3 := bProgram3_On;
INDEXING_1_VAR.DataByteOutput[0].4 := bProgram4_On;
INDEXING_1_VAR.DataByteOutput[0].6 := bResetInput;
INDEXING_1_VAR.DataByteOutput[0].7 := bHomePositionReturn;
INDEXING_1_VAR.DataByteOutput[1].0 := bStartInput;
INDEXING_1_VAR.DataByteOutput[1].1 := bServoOn;
INDEXING_1_VAR.DataByteOutput[1].2 := bFirstDigit;
INDEXING_1_VAR.DataByteOutput[1].4 := bEmergencyInput;

IN_POSITION_INPUT := 			INDEXING_1_VAR.DataByteInput [1].0;
IN_POSITIONING_COMPLETION := 	INDEXING_1_VAR.DataByteInput [1].1;
IN_START_INPUT_WAIT := 			INDEXING_1_VAR.DataByteInput [1].2;
IN_ALARM1 := 					INDEXING_1_VAR.DataByteInput [1].3;
IN_ALARM2 := 					INDEXING_1_VAR.DataByteInput [1].4;
IN_READY_STATE :=				INDEXING_1_VAR.DataByteInput [1].7;
IN_SERVO_STATUS :=				INDEXING_1_VAR.DataByteInput [1].6; 
(*
//SERVO ON
IF NOT IN_SERVO_STATUS THEN
	bResetInput := TRUE;
	TMR4(IN:=bResetInput,PT:=T#0.5S);
	IF TMR4.Q THEN
		bResetInput := FALSE;
	END_IF
	bServoOn:=TRUE;
	//POWER_CONTROL.O_PWR_CTRL_INDEXING_1:=TRUE;
	TMR8(IN:=POWER_CONTROL.O_PWR_CTRL_INDEXING_1,PT:=T#0.5S);	
	IF TMR8.Q THEN
		POWER_CONTROL.O_PWR_CTRL_INDEXING_1:=FALSE;
		TMR8(IN:=FALSE);
	END_IF
END_IF
*)
//ALARM RESET
IF NOT IN_ALARM1 OR NOT IN_ALARM2 THEN
	bResetInput := TRUE;
	TMR4(IN:=bResetInput,PT:=T#0.5S);
	INPUT_VAR.ALARM1:=NOT IN_ALARM1 OR NOT IN_ALARM2;
	IF TMR4.Q THEN
		bResetInput := FALSE;
	END_IF
ELSE
	TMR4(IN:=FALSE);
END_IF

IF INDEXING_1_VAR.I_INDEXING_1_ROTATION_DONE THEN
		INDEXING_1_VAR.I_INDEXING_1_HOME:=TRUE;
		bHomePositionReturn:=FALSE;
		//INDEXING_1_VAR.I_INDEXING_1_ROTATION_DONE:=TRUE;
END_IF
//homing
IF NOT INDEXING_1_VAR.I_INDEXING_1_HOME THEN
	bHomePositionReturn:=TRUE;
 	ResetCount:=TRUE;
	INDEXING_1_VAR.O_ROTATION_START:=FALSE;
	INDEXING_1_VAR.I_INDEXING_1_ROTATION_DONE:=FALSE;
	
	INPUT_G6_VAR.O_G6_GRIPPER_EXT_DOWN_1:=FALSE;
	INPUT_G6_VAR.O_G6_GRIPPER_EXT_UP_1:=TRUE;
	
	INPUT_G6_VAR.O_G6_GRIPPER_EXT_DOWN_2:=FALSE;
	INPUT_G6_VAR.O_G6_GRIPPER_EXT_UP_2:=TRUE;
	
	INPUT_G6_VAR.O_G6_GRIPPER_EXT_DOWN_3:=FALSE;
	INPUT_G6_VAR.O_G6_GRIPPER_EXT_UP_3:=TRUE;
	
	INPUT_G6_VAR.O_G6_GRIPPER_EXT_DOWN_4:=FALSE;
	INPUT_G6_VAR.O_G6_GRIPPER_EXT_UP_4:=TRUE;
END_IF



IF (bHomePositionReturn OR bprogram0_on) AND NOT INDEXING_1_VAR.I_INDEXING_1_ROTATION_DONE THEN
	TMR_OFF(IN:=TRUE,PT:=T#40S);
	IF TMR_OFF.Q THEN
		POWER_CONTROL.O_PWR_CTRL_INDEXING_1:=TRUE;
		TMR_RELEASE(IN:=TRUE,PT:=T#0.5S);
		bHomePositionReturn:=FALSE;
	
	END_IF
ELSE
	TMR_OFF(IN:=FALSE);
	TMR_RELEASE(IN:=FALSE);
END_IF
IF TMR_RELEASE.Q THEN
	POWER_CONTROL.O_PWR_CTRL_INDEXING_1:=FALSE;
	TMR_OFF(IN:=FALSE);
END_IF
//start indexing
START_ROTATING(CLK:=INDEXING_1_VAR.O_ROTATION_START);
IF INDEXING_1_VAR.O_ROTATION_START AND IN_START_INPUT_WAIT AND INDEXING_1_VAR.I_INDEXING_1_HOME AND INPUT_VAR.STRAIGHTEN_DONE  THEN
	INDEXING_1_VAR.READY_STRAIGTHEN:=TRUE;
	ELSE
	INDEXING_1_VAR.READY_STRAIGTHEN:=FALSE;	
END_IF

START_ROTATION(IN:=INDEXING_1_VAR.READY_STRAIGTHEN,PT:=T#0.5S);
IF 	START_ROTATION.Q AND NOT TMR_PROCESS.Q AND INDEXING_1_VAR.I_PRESS_STOPPER_UP AND NOT INPUT_G6_VAR.I_G6_START_PLACING AND NOT LOADER_RS4_VAR.I_LOADER_RS4_START_TAKEUP AND INPUT_VAR.STRAIGHTEN_DONE AND NOT INPUT_G6_VAR.I_G6_START_PLACING AND NOT LOADER_RS4_VAR.I_LOADER_RS4_START_TAKEUP THEN
	bprogram0_on:=TRUE;
	IF bprogram0_on THEN
		INDEXING_1_VAR.O_ROTATION_START:=FALSE;
	END_IF
	INDEXING_1_VAR.I_INDEXING_1_ROTATION_DONE:=FALSE;
	IN_POSITIONING_COMPLET :=FALSE;
END_IF
IF bprogram0_on THEN
		A:=FALSE;
	TMR_PROCESS(IN:=TRUE,PT:=T#3S);
	INDEXING_1_VAR.O_ROTATION_START:=FALSE;
	INDEXING_1_VAR.I_INDEXING_1_ROTATION_DONE:=FALSE;
ELSE
	TMR_PROCESS(IN:=FALSE);
END_IF
//select Program No.
IF bprogram0_on AND INDEXING_1_VAR.I_PRESS_STOPPER_UP AND NOT INPUT_G6_VAR.I_G6_START_PLACING AND NOT LOADER_RS4_VAR.I_LOADER_RS4_START_TAKEUP  THEN
	TMR1(IN:=bprogram0_on,PT:=T#15MS);
	bStartInput:=tmr1.Q ;
	IF tmr1.Q THEN
		TMR2(in:=TRUE,pt:=T#25MS);
	END_IF
	IF tmr2.Q THEN
		tmr1(in:=FALSE);
		bStartInput:=FALSE;
	END_IF
	tmr3(in:=tmr2.Q,pt:=T#5MS);
	IF tmr3.Q THEN
		bprogram0_on:= FALSE;
		tmr2(in:=FALSE);
		tmr3(in:=FALSE);
	END_IF
END_IF

IPC(IN:=IN_POSITIONING_COMPLETION,PT:=T#0.01S);
INPOS(CLK:=IN_POSITIONING_COMPLETION);
IF INPOS.Q OR  IN_POSITIONING_COMPLETION THEN
	A:=TRUE;
	IN_POSITIONING_COMPLET :=TRUE;
	INDEXING_1_VAR.I_INDEXING_1_ROTATION_DONE:=TRUE;
END_IF
IF A THEN
	IN_POSITIONING_COMPLET :=TRUE;
	INDEXING_1_VAR.I_INDEXING_1_ROTATION_DONE:=TRUE;
END_IF
IF 	IN_POSITIONING_COMPLET THEN
	INDEXING_1_VAR.I_INDEXING_1_ROTATION_DONE:=TRUE;
END_IF
//IF INDEXING_1_VAR.I_PRESS_STOPPER_UP AND INDEXING_1_VAR.I_INDEXING_1_ROTATION_DONE THEN
IF INDEXING_1_VAR.I_INDEXING_1_ROTATION_DONE THEN
	SS(CLK:=INDEXING_1_VAR.I_INDEXING_1_ROTATION_DONE );
	CNT_START(CU:=SS.Q,RESET:= CNT_START.Q,PV:=2);
	IN_POSITIONING_COMPLET :=FALSE;
	//IF CNT_START.CV=1 THEN
		INPUT_VAR.STRAIGHTEN_START:=SS.Q;
	//END_IF
ELSE
	SS(CLK:=FALSE);
END_IF

IF INPUT_G6_VAR.I_G6_START_PLACING OR LOADER_RS4_VAR.I_LOADER_RS4_START_TAKEUP THEN
	bprogram0_on:= FALSE;
	bStartInput:=FALSE;
END_IF

END_PROGRAM

// ---- POUs/LOADER/INDEX_1.TcPOU
PROGRAM INDEX_1
VAR
	bStartInput : BOOL;
	bServoOn : BOOL;
	bProgram0_On : BOOL;
	bProgram1_On : BOOL :=TRUE;
	bProgram2_On : BOOL :=FALSE;
	bProgram3_On : BOOL:=FALSE;
	bProgram4_On : BOOL:=FALSE;	
	bHomePositionReturn : BOOL;
	bResetInput : BOOL;
	bEmergencyInput : BOOL := TRUE;
	
	IN_POSITION_INPUT: BOOL;
	IN_POSITIONING_COMPLETION: BOOL;
	IN_START_INPUT_WAIT: BOOL;
	IN_ALARM1: BOOL;
	IN_ALARM2: BOOL;
	IN_READY_STATE: BOOL;
	T1: TON;
	TMR1: TON;
	TMR2: TON;
	TMR3: TON;
	TMR4: TON;
	TMR5: TON;
	TMR6: TON;
	TMR7: TON;
	IN_SERVO_STATUS: BOOL;
	bFirstDigit: BOOL;
	CNT1: CTU;
	ResetCount: BOOL;
	IPC: TP;
	IN_POSITIONING_COMPLET: BOOL;
	CNT2: CTU;
	START_STRAIGTHEN: BOOL;

	START_STRAIGHTEN: R_TRIG;
	START_ROTATING: R_TRIG;
	START_ROTATION: TP;
	SS: R_TRIG;
	CNT_START: CTU;
	TMR_PROCESS: TOF;
END_VAR

INDEXING_1_VAR.DataByteOutput[0].0 := bProgram0_On;
INDEXING_1_VAR.DataByteOutput[0].1 := bProgram1_On;
INDEXING_1_VAR.DataByteOutput[0].2 := bProgram2_On;
INDEXING_1_VAR.DataByteOutput[0].3 := bProgram3_On;
INDEXING_1_VAR.DataByteOutput[0].4 := bProgram4_On;
INDEXING_1_VAR.DataByteOutput[0].6 := bResetInput;
INDEXING_1_VAR.DataByteOutput[0].7 := bHomePositionReturn;
INDEXING_1_VAR.DataByteOutput[1].0 := bStartInput;
INDEXING_1_VAR.DataByteOutput[1].1 := bServoOn;
INDEXING_1_VAR.DataByteOutput[1].2 := bFirstDigit;
INDEXING_1_VAR.DataByteOutput[1].4 := bEmergencyInput;

IN_POSITION_INPUT := 			INDEXING_1_VAR.DataByteInput [1].0;
IN_POSITIONING_COMPLETION := 	INDEXING_1_VAR.DataByteInput [1].1;
IN_START_INPUT_WAIT := 			INDEXING_1_VAR.DataByteInput [1].2;
IN_ALARM1 := 					INDEXING_1_VAR.DataByteInput [1].3;
IN_ALARM2 := 					INDEXING_1_VAR.DataByteInput [1].4;
IN_READY_STATE :=				INDEXING_1_VAR.DataByteInput [1].7;
IN_SERVO_STATUS :=				INDEXING_1_VAR.DataByteInput [1].6; 

//ALARM RESET
IF IN_ALARM1 OR IN_ALARM2 THEN
	bResetInput := TRUE;
	TMR4(IN:=bResetInput,PT:=T#0.5S);
	IF TMR4.Q THEN
		bResetInput := FALSE;
	END_IF
ELSE
	TMR4(IN:=FALSE);
END_IF

IF NOT INDEXING_1_VAR.I_INDEXING_1_HOME THEN
	INDEXING_1_VAR.O_INDEXING_1_HOME:=TRUE;
 	ResetCount:=TRUE;
	INDEXING_1_VAR.O_ROTATION_START:=FALSE;
 	IF IN_POSITIONING_COMPLET THEN
		INDEXING_1_VAR.I_INDEXING_1_HOME:=TRUE;
	END_IF
END_IF

IF INDEXING_1_VAR.O_INDEXING_1_HOME THEN
	bHomePositionReturn:=TRUE;
	IF IN_POSITIONING_COMPLET THEN
		INDEXING_1_VAR.O_INDEXING_1_HOME:=FALSE;
		bHomePositionReturn:=FALSE;
	END_IF
END_IF

START_ROTATION(IN:=INDEXING_1_VAR.O_ROTATION_START,PT:=T#0.1S);
IF 	START_ROTATION.Q AND NOT TMR_PROCESS.Q THEN
	bprogram0_on:=TRUE;
	IF bprogram0_on THEN
		INDEXING_1_VAR.O_ROTATION_START:=FALSE;
	END_IF
	
	INDEXING_1_VAR.I_INDEXING_1_ROTATION_DONE:=FALSE;
	IN_POSITIONING_COMPLET :=FALSE;
END_IF
IF bprogram0_on THEN
	TMR_PROCESS(IN:=TRUE,PT:=T#3S);
	INDEXING_1_VAR.O_ROTATION_START:=FALSE;
ELSE
	TMR_PROCESS(IN:=FALSE);
END_IF
//select Program No.
IF bprogram0_on   THEN
	INDEXING_1_VAR.O_ROTATION_START:=FALSE;
	TMR1(IN:=bprogram0_on,PT:=T#15MS);
	bStartInput:=tmr1.Q ;
	IF tmr1.Q THEN
		TMR2(in:=TRUE,pt:=T#25MS);
	END_IF
	
	IF tmr2.Q THEN
		tmr1(in:=FALSE);
		bStartInput:=FALSE;
	END_IF
	tmr3(in:=tmr2.
Q,pt:=T#5MS);
	IF tmr3.Q THEN
		bprogram0_on:= FALSE;
		tmr2(in:=FALSE);
		tmr3(in:=FALSE);
	END_IF
END_IF

IPC(IN:=IN_POSITIONING_COMPLETION,PT:=T#0.4S);
IF IPC.Q THEN
	IN_POSITIONING_COMPLET :=TRUE;
END_IF
IF 	IN_POSITIONING_COMPLET THEN
	INDEXING_1_VAR.I_INDEXING_1_ROTATION_DONE:=TRUE;
END_IF
IF INDEXING_1_VAR.I_PRESS_STOPPER_UP AND INDEXING_1_VAR.I_INDEXING_1_ROTATION_DONE THEN
	SS(CLK:=INDEXING_1_VAR.I_INDEXING_1_ROTATION_DONE );
	CNT_START(CU:=SS.Q,RESET:= CNT_START.Q,PV:=2);
	IF CNT_START.CV=1 THEN
	INPUT_VAR.STRAIGHTEN_START:=SS.Q;
	END_IF
	IN_POSITIONING_COMPLET :=FALSE;
	ELSE
SS(CLK:=FALSE);
END_IF

END_PROGRAM

// ---- POUs/LOADER/INDEXING_2.TcPOU
PROGRAM INDEXING_2
VAR
	bStartInput : BOOL;
	bServoOn : BOOL;
	bProgram0_On : BOOL;
	bProgram1_On : BOOL :=TRUE;
	bProgram2_On : BOOL :=FALSE;
	bProgram3_On : BOOL:=FALSE;
	bProgram4_On : BOOL:=FALSE;	
	bHomePositionReturn : BOOL;
	bResetInput : BOOL;
	bEmergencyInput : BOOL := TRUE;
	
	IN_POSITION_INPUT: BOOL;
	IN_POSITIONING_COMPLETION: BOOL;
	IN_START_INPUT_WAIT: BOOL;
	IN_ALARM1: BOOL;
	IN_ALARM2: BOOL;
	IN_READY_STATE: BOOL;
	T1: TON;
	TMR1: TON;
	TMR2: TON;
	TMR3: TON;
	TMR4: TON;
	TMR5: TON;
	TMR6: TON;
	TMR7: TON;
	IN_SERVO_STATUS: BOOL;
	CNT1: CTU;
	ENABLE_TIMER: INT;
	ResetCount: BOOL;
	CNT_INDEX: CTU;
	
	RESET_CNT_INDEX: BOOL;
	TMR8: TON;
	M1:BOOL;
	M2:BOOL;
	M3:BOOL;
	M4:BOOL;
	TMR_OFF: TON;
	TMR_RELEASE: TON;
	IDX: INT;
END_VAR

VAR CONSTANT
	ISP: R_TRIG;
END_VAR

INDEXING_2_VAR.DataByteOutput2[0].0 := bProgram0_On;
INDEXING_2_VAR.DataByteOutput2[0].1 := bProgram1_On;
INDEXING_2_VAR.DataByteOutput2[0].2 := bProgram2_On;
INDEXING_2_VAR.DataByteOutput2[0].3 := bProgram3_On;
INDEXING_2_VAR.DataByteOutput2[0].4 := bProgram4_On;
INDEXING_2_VAR.DataByteOutput2[0].6 := bResetInput;
INDEXING_2_VAR.DataByteOutput2[0].7 := bHomePositionReturn;
INDEXING_2_VAR.DataByteOutput2[1].0 := bStartInput;
INDEXING_2_VAR.DataByteOutput2[1].1 := bServoOn;
INDEXING_2_VAR.DataByteOutput2[1].4 := bEmergencyInput;

IN_POSITION_INPUT := INDEXING_2_VAR.DataByteInput2 [1].0;
IN_POSITIONING_COMPLETION := INDEXING_2_VAR.DataByteInput2 [1].1;
IN_START_INPUT_WAIT := INDEXING_2_VAR.DataByteInput2 [1].2;
IN_ALARM1 := INDEXING_2_VAR.DataByteInput2 [1].3;
IN_ALARM2 := INDEXING_2_VAR.DataByteInput2 [1].4;
IN_READY_STATE :=INDEXING_2_VAR.DataByteInput2 [1].7;
IN_SERVO_STATUS :=INDEXING_2_VAR.DataByteInput2 [1].6; 

M1:=INDEXING_2_VAR.DataByteInput2 [0].0;
M2:=INDEXING_2_VAR.DataByteInput2 [0].1;
M3:=INDEXING_2_VAR.DataByteInput2 [0].2;
M4:=INDEXING_2_VAR.DataByteInput2 [0].3;
bProgram1_On:=FALSE;
bProgram2_On:=FALSE;
bProgram3_On:=FALSE;
bProgram4_On:=FALSE;

//CEK SERVO STATUS
IF NOT IN_SERVO_STATUS THEN
	bResetInput := TRUE;
	TMR4(IN:=bResetInput,PT:=T#0.5S);
	IF TMR4.Q THEN
		bResetInput := FALSE;
	END_IF
	bServoOn:=TRUE;
	//POWER_CONTROL.O_PWR_CTRL_INDEXING_2:=TRUE;
	TMR8(IN:=POWER_CONTROL.O_PWR_CTRL_INDEXING_2,PT:=T#0.5S);	
	IF TMR8.Q THEN
		POWER_CONTROL.O_PWR_CTRL_INDEXING_2:=FALSE;
		TMR8(IN:=FALSE);
	END_IF
END_IF

//ALARM RESET
IF NOT IN_ALARM1 OR NOT IN_ALARM2 THEN
	bResetInput := TRUE;
	TMR4(IN:=bResetInput,PT:=T#0.5S);
		INPUT_VAR.ALARM1:=NOT IN_ALARM1 OR NOT IN_ALARM2;
	IF TMR4.Q THEN
		bResetInput := FALSE;
	END_IF
ELSE
	TMR4(IN:=FALSE);
END_IF

//HOMING
IF NOT INDEXING_2_VAR.I_INDEXING_2_HOME THEN
 	INDEXING_2_VAR.O_INDEXING_HOME:=TRUE;
END_IF
 
IF INDEXING_2_VAR.O_INDEXING_HOME THEN
	bHomePositionReturn:=TRUE;
	ResetCount:=TRUE;
	INDEXING_2_VAR.I_INDEXING_2_ROTATION_DONE:=FALSE;
	RESET_CNT_INDEX:=TRUE;
ELSE
	RESET_CNT_INDEX:=FALSE;
	bHomePositionReturn:=FALSE;
END_IF

ISP(CLK:=IN_POSITIONING_COMPLETION);	
IF 	ISP.Q THEN
	INDEXING_2_VAR.I_INDEXING_2_ROTATION_DONE:=TRUE;
END_IF

IF INDEXING_2_VAR.I_INDEXING_2_ROTATION_DONE OR INDEXING_2_VAR.O_ROTATION_DONE THEN
	INDEXING_2_VAR.I_INDEXING_2_HOME:=TRUE;
	INDEXING_2_VAR.O_INDEXING_HOME:=FALSE;
END_IF
//POWER RESET
IF bHomePositionReturn OR NOT INDEXING_2_VAR.I_INDEXING_2_ROTATION_DONE THEN
	TMR_OFF(IN:=TRUE,PT:=T#60S);
	IF TMR_OFF.Q THEN
		POWER_CONTROL.O_PWR_CTRL_INDEXING_2:=TRUE;
		TMR_RELEASE(IN:=TRUE,PT:=T#0.5S);
		BPROGRAM0_ON:=FALSE;
	END_IF
ELSE
	TMR_OFF(IN:=FALSE);
	TMR_RELEASE(IN:=FALSE);
END_IF

IF TMR_RELEASE.Q THEN
	POWER_CONTROL.O_PWR_CTRL_INDEXING_1:=FALSE;
	TMR_OFF(IN:=FALSE);
END_IF



//START ROTATION 
	IF 	INDEXING_2_VAR.O_ROTATION_START AND IN_START_INPUT_WAIT AND NOT INDEXING_2_VAR.O_INDEXING_HOME THEN
		IDX:=1;
		INDEXING_2_VAR.I_INDEXING_2_ROTATION_DONE:=FALSE;
	END_IF
CASE IDX OF
1:
	bprogram0_on:=TRUE;
	IF BPROGRAM0_ON THEN
		IDX:=2;
		INDEXING_2_VAR.O_ROTATION_START:=FALSE;
	END_IF

2:
//select Program No.
	IF bprogram0_on THEN
		INDEXING_2_VAR.O_ROTATION_START:=FALSE;
		INDEXING_2_VAR.I_INDEXING_2_ROTATION_DONE:=FALSE;
		TMR1(IN:=bprogram0_on,PT:=T#15MS);
		bStartInput:=tmr1.Q ;
		IF tmr1.Q THEN
			TMR2(in:=TRUE,pt:=T#25MS);
		END_IF
	
		IF tmr2.Q THEN
			tmr1(in:=FALSE);
			bStartInput:=FALSE;
		END_IF
		tmr3(in:=tmr2.Q,pt:=T#5MS);
		IF tmr3.Q THEN
			bprogram0_on:= FALSE;
			tmr2(in:=FALSE);
			tmr3(in:=FALSE);
			
		END_IF
	END_IF
	IF 	ISP.Q THEN
		INDEXING_2_VAR.O_ROTATION_DONE:=TRUE;
		INDEXING_2_VAR.O_ROTATION_START:=FALSE;
		INDEXING_2_VAR.I_INDEXING_2_ROTATION_DONE:=TRUE;
		IDX:=3;
	END_IF
3:
		IF INDEXING_2_VAR.I_INDEXING_2_ROTATION_DONE OR INDEXING_2_VAR.O_ROTATION_DONE THEN
		IDX:=0;
	END_IF	
END_CASE


IF  INDEXING_2_VAR.I_INDEXING_2_HOME THEN
	CNT_INDEX(CU:=bprogram0_on,RESET:=CNT_INDEX.Q,PV:=4);
	ELSE
	CNT_INDEX(CU:=FALSE);
	INDEXING_2_VAR.CARRIER_INDEX :=100;
END_IF

CASE CNT_INDEX.CV OF
	0:
	INDEXING_2_VAR.CARRIER_INDEX :=0;
	RESET_CNT_INDEX:=FALSE;
	1:
	INDEXING_2_VAR.CARRIER_INDEX :=1;
	2:
	INDEXING_2_VAR.CARRIER_INDEX :=2;
	3:
	INDEXING_2_VAR.CARRIER_INDEX :=3;
ELSE
	INDEXING_2_VAR.CARRIER_INDEX :=0;
END_CASE

IF RESET_CNT_INDEX THEN
	CNT_INDEX(CU:=FALSE);
END_IF
//START ROTATING TRIGGER BY 3 ROBOTS
IF (TESTER_C8_VAR.READY_INDEXING AND LOADER_RS4_VAR.READY_INDEXING AND SORTER_RS4_VAR.READY_INDEXING)
	OR (LOADER_RS4_VAR.READY_INDEXING AND NOT TESTER_C8_VAR.O_C8_ENABLE)
	OR (TESTER_C8_VAR.READY_INDEXING AND LOADER_RS4_VAR.READY_INDEXING AND NOT SORTER_RS4_VAR.I_SORTER_RS4_ENABLE) THEN
	INDEXING_2_VAR.O_ROTATION_START:=TRUE;
ELSE
	INDEXING_2_VAR.O_ROTATION_START:=FALSE;
END_IF

END_PROGRAM

// ---- POUs/LOADER/STRAIGHTENING_PROG_1.TcPOU
 PROGRAM STRAIGHTENING_PROG_1
VAR

	NEW: INT;
	FG: INT;
	ENABLE_TIMER: BOOL := FALSE;
	TMR1: TON;
	TMR2: TON;
	CNT1: CTU;
END_VAR

IF INPUT_VAR.STRAIGHTEN_START AND INDEXING_1_VAR.I_INDEXING_1_ROTATION_DONE THEN
	ENABLE_TIMER:=TRUE;
END_IF
IF ENABLE_TIMER THEN
	INPUT_VAR.STRAIGHTEN_START:=FALSE;
	TMR1(IN:=NOT TMR2.Q,PT:=T#0.15S);
	TMR2(IN:=TMR1.Q,PT:=T#0.3S);
	IF TMR2.Q THEN
		TMR1(IN:=FALSE); 
		TMR2(IN:=FALSE);
	END_IF
	
	(*IF NOT  INDEXING_1_VAR.I_PRESS_STOPPER_DOWN  THEN
		INDEXING_1_VAR.O_PRESS_STOPPER_DOWN:=TRUE;
		INDEXING_1_VAR.O_PRESS_STOPPER_UP:=FALSE;
	END_IF*)
ELSE
		TMR1(IN:=FALSE);
		TMR2(IN:=FALSE);
END_IF

CNT1(CU:=TMR1.Q,RESET:=NOT	ENABLE_TIMER,PV:=10);
//CNT1(CU:=TMR1.Q,RESET:=NOT INPUT_VAR.STRAIGHTEN_START,PV:=11);
IF CNT1.CV >=12 THEN
	ENABLE_TIMER:=FALSE;
	INDEXING_1_VAR.STRAIGHTEN_FINISH:=TRUE;
	INDEXING_1_VAR.O_PRESS_STOPPER_DOWN:=FALSE;
	INDEXING_1_VAR.O_PRESS_STOPPER_UP:=TRUE;
END_IF

IF CNT1.CV =2 THEN
	INDEXING_1_VAR.STRAIGHTEN_FINISH:=FALSE;
END_IF

IF 	INDEXING_1_VAR.STRAIGHTEN_FINISH THEN
	IF INDEXING_1_VAR.I_PRESS_STOPPER_UP THEN
		INPUT_VAR.STRAIGHTEN_DONE :=TRUE;	
		INPUT_VAR.STRAIGHTEN_PROCESS:=FALSE;
	END_IF	
END_IF
CASE CNT1.CV OF	
//CASE INDEXING_1_VAR.INDEXING_1_CASE OF
0:	
	INDEXING_1_VAR.O_PRESS_STOPPER_DOWN:=FALSE;
	INDEXING_1_VAR.O_PRESS_STOPPER_UP:=TRUE;
	INDEXING_1_VAR.I_INDEXING_1_READY_FOR_STRAIGHTEN:=FALSE;

1: 	INDEXING_1_VAR.O_PRESS_STOPPER_DOWN:=TRUE;
	INDEXING_1_VAR.O_PRESS_STOPPER_UP:=FALSE;

2: 	INDEXING_1_VAR.O_PRESS_STOPPER_DOWN:=TRUE;
	INDEXING_1_VAR.O_PRESS_STOPPER_UP:=FALSE;
	
3: 	INDEXING_1_VAR.O_PRESS_STOPPER_DOWN:=FALSE;
	INDEXING_1_VAR.O_PRESS_STOPPER_UP:=TRUE;
	
4: 	INDEXING_1_VAR.O_PRESS_STOPPER_DOWN:=TRUE;
	INDEXING_1_VAR.O_PRESS_STOPPER_UP:=FALSE;
5:	
	INPUT_VAR.STRAIGHTEN_PROCESS:=TRUE;
	INDEXING_1_VAR.O_INDEXING_1_GRIPPER_OPEN_1:=TRUE;
	INDEXING_1_VAR.O_INDEXING_1_GRIPPER_CLOSE_1:=FALSE;
		
6:
	INDEXING_1_VAR.O_INDEXING_1_GRIPPER_EXT_UP :=TRUE;	
	INDEXING_1_VAR.O_INDEXING_1_GRIPPER_EXT_down:=FALSE;
		
7:
	INDEXING_1_VAR.O_INDEXING_1_GRIPPER_OPEN_1:=FALSE;
	INDEXING_1_VAR.O_INDEXING_1_GRIPPER_CLOSE_1:=TRUE;
	//INDEXING_1_VAR.O_PRESS_STOPPER_DOWN:=FALSE;
	//INDEXING_1_VAR.O_PRESS_STOPPER_UP:=TRUE;		
8:
	INDEXING_1_VAR.O_INDEXING_1_GRIPPER_EXT_UP :=FALSE;	
	INDEXING_1_VAR.O_INDEXING_1_GRIPPER_EXT_down:=TRUE;
	
9:	
	INDEXING_1_VAR.O_INDEXING_1_GRIPPER_OPEN_1:=TRUE;
	INDEXING_1_VAR.O_INDEXING_1_GRIPPER_CLOSE_1:=FALSE;
	//INDEXING_1_VAR.O_PRESS_STOPPER_DOWN:=TRUE;
	//INDEXING_1_VAR.O_PRESS_STOPPER_UP:=FALSE;	
10:
	INDEXING_1_VAR.O_INDEXING_1_GRIPPER_EXT_UP :=TRUE;	
	INDEXING_1_VAR.O_INDEXING_1_GRIPPER_EXT_down:=FALSE;	
11:
	INDEXING_1_VAR.O_INDEXING_1_GRIPPER_OPEN_1:=FALSE;
	INDEXING_1_VAR.O_INDEXING_1_GRIPPER_CLOSE_1:=TRUE;
			
12:
	INDEXING_1_VAR.O_INDEXING_1_GRIPPER_EXT_UP :=FALSE;	
	INDEXING_1_VAR.O_INDEXING_1_GRIPPER_EXT_down:=TRUE;
	ENABLE_TIMER:=FALSE;
	INPUT_VAR.STRAIGHTEN_START:=FALSE;
END_CASE

IF 
	INDEXING_1_VAR.O_INDEXING_1_GRIPPER_OPEN_1 AND
	INDEXING_1_VAR.I_INDEXING_1_GRIPPER_OPEN_1 AND
	INDEXING_1_VAR.I_INDEXING_1_GRIPPER_OPEN_2	AND
	INDEXING_1_VAR.I_INDEXING_1_GRIPPER_OPEN_3	AND 
	INDEXING_1_VAR.I_INDEXING_1_GRIPPER_OPEN_4	AND
	NOT INDEXING_1_VAR.I_INDEXING_1_GRIPPER_CLOSE_1	AND
	NOT INDEXING_1_VAR.I_INDEXING_1_GRIPPER_CLOSE_2	AND
	NOT INDEXING_1_VAR.I_INDEXING_1_GRIPPER_CLOSE_3	AND
	NOT INDEXING_1_VAR.I_INDEXING_1_GRIPPER_CLOSE_4 THEN
		INDEXING_1_VAR.I_ALL_GRIPPER_OPEN :=TRUE;
	END_IF

IF 
	NOT INDEXING_1_VAR.O_INDEXING_1_GRIPPER_OPEN_1 AND
	NOT INDEXING_1_VAR.I_INDEXING_1_GRIPPER_OPEN_1 AND
	NOT INDEXING_1_VAR.I_INDEXING_1_GRIPPER_OPEN_2	AND
	NOT INDEXING_1_VAR.I_INDEXING_1_GRIPPER_OPEN_3	AND 
	NOT INDEXING_1_VAR.I_INDEXING_1_GRIPPER_OPEN_4	AND
	INDEXING_1_VAR.I_INDEXING_1_GRIPPER_CLOSE_1	AND
	INDEXING_1_VAR.I_INDEXING_1_GRIPPER_CLOSE_2	AND
	INDEXING_1_VAR.I_INDEXING_1_GRIPPER_CLOSE_3	AND
	INDEXING_1_VAR.I_INDEXING_1_GRIPPER_CLOSE_4 THEN
		INDEXING_1_VAR.I_ALL_GRIPPER_OPEN :=FALSE;
END_IF


	INDEXING_1_VAR.O_INDEXING_1_GRIPPER_OPEN_2:=INDEXING_1_VAR.O_INDEXING_1_GRIPPER_OPEN_1;
	INDEXING_1_VAR.O_INDEXING_1_GRIPPER_OPEN_3:=INDEXING_1_VAR.O_INDEXING_1_GRIPPER_OPEN_1;
	INDEXING_1_VAR.O_INDEXING_1_GRIPPER_OPEN_4:=INDEXING_1_VAR.O_INDEXING_1_GRIPPER_OPEN_1;

	INDEXING_1_VAR.O_INDEXING_1_GRIPPER_CLOSE_2:=INDEXING_1_VAR.O_INDEXING_1_GRIPPER_CLOSE_1;
	INDEXING_1_VAR.O_INDEXING_1_GRIPPER_CLOSE_3:=INDEXING_1_VAR.O_INDEXING_1_GRIPPER_CLOSE_1;
	INDEXING_1_VAR.O_INDEXING_1_GRIPPER_CLOSE_4:=INDEXING_1_VAR.O_INDEXING_1_GRIPPER_CLOSE_1;

END_PROGRAM

// ---- POUs/ROBOT/INPUT_G6.TcPOU
PROGRAM INPUT_G6
VAR
	TMR11: TON;
	TMR12: TON;
	TMR10: TON;
	TMR8: TON;
	TMR9: TON;
	TMR7: TON;
	TMR3: TON;
	TP1: TP;
	TMR1: TON;
	START_ROBOT: TP;
	TP2: TP;
	O_G6_HANG: BOOL;
	I_G6_HANG: BOOL;
	TMR2: TON;
	GO_ROBOT: BOOL;
	TP3: TP;
	TMR4: TON;
	CNT_CYCLE: CTU;
	START_ROTATE: R_TRIG;
	IN: INT;
	TP_END_FUKUDA: TP;
	CNT_END_FUKUDA: CTU;
	ROBOT_READY: BOOL;
	ROBOT_G6_READY: BOOL;
	END_FUKUDA: BOOL;
	O_END_FUKUDA: BOOL;
	TEMP_COUNTER_FUKUDA_A: INT;
	TEMP_COUNTER_FUKUDA_B: INT;
	O_END_FUKUDB: BOOL;
	MAX_DEVICE: INT;
	TMR_HANG: TON;
	GRP1: Tp;
	GRP2: Tp;
	GRP3: Tp;
	GRP4: Tp;
	CNT_PLACING: ctu;
	CNT_TAKING: CTU;
	CNT_CYCLE1: CTU;
END_VAR

VAR PERSISTENT
	TRGEN: R_TRIG;
END_VAR

IF INPUT_G6_VAR.I_G6_ENABLE  THEN
//GRIPPING 
IF INPUT_G6_VAR.IX_G6_GRIPPER_1 THEN
	INPUT_G6_VAR.O_G6_GRIPPER_CLOSE_1:=TRUE;
	INPUT_G6_VAR.O_G6_GRIPPER_OPEN_1:=FALSE;
ELSE
	INPUT_G6_VAR.O_G6_GRIPPER_CLOSE_1:=FALSE;
	INPUT_G6_VAR.O_G6_GRIPPER_OPEN_1:=TRUE;
END_IF

IF INPUT_G6_VAR.IX_G6_GRIPPER_2 THEN
	INPUT_G6_VAR.O_G6_GRIPPER_CLOSE_2:=TRUE;
	INPUT_G6_VAR.O_G6_GRIPPER_OPEN_2:=FALSE;
ELSE
	INPUT_G6_VAR.O_G6_GRIPPER_CLOSE_2:=FALSE;
	INPUT_G6_VAR.O_G6_GRIPPER_OPEN_2:=TRUE;
END_IF 

IF INPUT_G6_VAR.IX_G6_GRIPPER_3 THEN
	INPUT_G6_VAR.O_G6_GRIPPER_CLOSE_3:=TRUE;
	INPUT_G6_VAR.O_G6_GRIPPER_OPEN_3:=FALSE;
ELSE
	INPUT_G6_VAR.O_G6_GRIPPER_CLOSE_3:=FALSE;
	INPUT_G6_VAR.O_G6_GRIPPER_OPEN_3:=TRUE;
END_IF

IF INPUT_G6_VAR.IX_G6_GRIPPER_4 THEN
	INPUT_G6_VAR.O_G6_GRIPPER_CLOSE_4:=TRUE;
	INPUT_G6_VAR.O_G6_GRIPPER_OPEN_4:=FALSE;
ELSE
	INPUT_G6_VAR.O_G6_GRIPPER_CLOSE_4:=FALSE;
	INPUT_G6_VAR.O_G6_GRIPPER_OPEN_4:=TRUE;
END_IF

//EXTENDER DOWN
IF INPUT_G6_VAR.IX_G6_GRIPPER_EXT_1 THEN
	INPUT_G6_VAR.O_G6_GRIPPER_EXT_DOWN_1:=TRUE;
	INPUT_G6_VAR.O_G6_GRIPPER_EXT_UP_1:=FALSE;
ELSE
	INPUT_G6_VAR.O_G6_GRIPPER_EXT_DOWN_1:=FALSE;
	INPUT_G6_VAR.O_G6_GRIPPER_EXT_UP_1:=TRUE;
END_IF

IF INPUT_G6_VAR.IX_G6_GRIPPER_EXT_2 THEN
	INPUT_G6_VAR.O_G6_GRIPPER_EXT_DOWN_2:=TRUE;
	INPUT_G6_VAR.O_G6_GRIPPER_EXT_UP_2:=FALSE;
ELSE
	INPUT_G6_VAR.O_G6_GRIPPER_EXT_DOWN_2:=FALSE;
	INPUT_G6_VAR.O_G6_GRIPPER_EXT_UP_2:=TRUE;
END_IF

IF INPUT_G6_VAR.IX_G6_GRIPPER_EXT_3 THEN
	INPUT_G6_VAR.O_G6_GRIPPER_EXT_DOWN_3:=TRUE;
	INPUT_G6_VAR.O_G6_GRIPPER_EXT_UP_3:=FALSE;
ELSE
	INPUT_G6_VAR.O_G6_GRIPPER_EXT_DOWN_3:=FALSE;
	INPUT_G6_VAR.O_G6_GRIPPER_EXT_UP_3:=TRUE;
END_IF

IF INPUT_G6_VAR.IX_G6_GRIPPER_EXT_4 THEN
	INPUT_G6_VAR.O_G6_GRIPPER_EXT_DOWN_4:=TRUE;
	INPUT_G6_VAR.O_G6_GRIPPER_EXT_UP_4:=FALSE;
ELSE
	INPUT_G6_VAR.O_G6_GRIPPER_EXT_DOWN_4:=FALSE;
	INPUT_G6_VAR.O_G6_GRIPPER_EXT_UP_4:=TRUE;
END_IF
IF INPUT_G6_VAR.I_G6_READY_TAKEUP THEN
	INPUT_G6_VAR.O_G6_GRIPPER_CLOSE_1:=FALSE;
	INPUT_G6_VAR.O_G6_GRIPPER_OPEN_1:=TRUE;
	
	INPUT_G6_VAR.O_G6_GRIPPER_CLOSE_2:=FALSE;
	INPUT_G6_VAR.O_G6_GRIPPER_OPEN_2:=TRUE;
	
	INPUT_G6_VAR.O_G6_GRIPPER_CLOSE_3:=FALSE;
	INPUT_G6_VAR.O_G6_GRIPPER_OPEN_3:=TRUE;
	
	INPUT_G6_VAR.O_G6_GRIPPER_CLOSE_3:=FALSE;
	INPUT_G6_VAR.O_G6_GRIPPER_OPEN_3:=TRUE;
END_IF

INPUT_G6_VAR.GRIPPER_OPEN_1:=INPUT_G6_VAR.I_G6_GRIPPER_OPEN_1;
INPUT_G6_VAR.GRIPPER_OPEN_2:=INPUT_G6_VAR.I_G6_GRIPPER_OPEN_2;
INPUT_G6_VAR.GRIPPER_OPEN_3:=INPUT_G6_VAR.I_G6_GRIPPER_OPEN_3;
INPUT_G6_VAR.GRIPPER_OPEN_4:=INPUT_G6_VAR.I_G6_GRIPPER_OPEN_4;

INPUT_G6_VAR.GRIPPER_CLOSE_1:=INPUT_G6_VAR.I_G6_GRIPPER_CLOSE_1;
INPUT_G6_VAR.GRIPPER_CLOSE_2:=INPUT_G6_VAR.I_G6_GRIPPER_CLOSE_2;
INPUT_G6_VAR.GRIPPER_CLOSE_3:=INPUT_G6_VAR.I_G6_GRIPPER_CLOSE_3;
INPUT_G6_VAR.GRIPPER_CLOSE_4:=INPUT_G6_VAR.I_G6_GRIPPER_CLOSE_4;

//ACTIVATE ROBOT
TRGEN(CLK:=INPUT_G6_VAR.I_G6_ENABLE); 
IF TRGEN.Q THEN
	INPUT_G6_VAR.O_G6_RESET_COUNTER_PICK:=TRUE;
END_IF
IF INPUT_G6_VAR.I_G6_START_PLACING OR INPUT_G6_VAR.I_G6_START_TAKEUP THEN
	INPUT_G6_VAR.O_G6_RESET_COUNTER_PICK:=FALSE;
END_IF
//IF INPUT_G6_VAR.I_G6_ENABLE THEN
TP_END_FUKUDA(IN:=INPUT_G6_VAR.I_G6_END_FUKUDA,PT:=T#0.1S);
CNT_END_FUKUDA(CU:=TP_END_FUKUDA.Q,RESET:=CNT_END_FUKUDA.Q,PV:=1000);

INPUT_VAR.I_STOPPER_TRANSFER_ON_A:= INPUT_VAR.O_STOPPER_TRANSFER_A;
//IF INPUT_VAR.I_STOPPER_TRANSFER_ON_A OR INPUT_VAR.I_STOPPER_TRANSFER_ON_B THEN
INPUT_G6_VAR.O_G6_SETMOTOROFF:=FALSE;
IF NOT INPUT_G6_VAR.I_G6_MOTORON THEN
	INPUT_G6_VAR.O_G6_STOP:=FALSE;
END_IF
IF NOT INPUT_G6_VAR.I_G6_MOTORON AND INPUT_G6_VAR.I_G6_READY AND NOT INPUT_G6_VAR.I_G6_ESTOPON AND NOT INPUT_G6_VAR.I_G6_SAFEGUARDON THEN
	INPUT_G6_VAR.O_G6_SETMOTORON:=TRUE;
	INPUT_G6_VAR.O_G6_STOP:=FALSE;
	INPUT_G6_VAR.O_G6_RESET :=FALSE;	
	INPUT_G6_VAR.O_G6_START :=FALSE ;
	INPUT_G6_VAR.O_G6_CONTINUE :=FALSE;
TMR1(IN:=INPUT_G6_VAR.O_G6_SETMOTORON ,PT:=T#0.5S);
ELSE
	INPUT_G6_VAR.O_G6_SETMOTOROFF:=FALSE;
	INPUT_G6_VAR.O_G6_SETMOTORON:=FALSE;
END_IF

//START POSITION CANNOT BE 0
IF INPUT_G6_VAR.START_POSITION =0 THEN
	INPUT_G6_VAR.START_POSITION :=1;
END_IF
// ERROR OVERRIDE	
	IF 	INPUT_G6_VAR.I_G6_ERROR OR INPUT_G6_VAR.I_CMDERROR THEN// AND INPUT_G6_VAR.I_G6_READY THEN// OR INPUT_G6_VAR.G6_ERROR1> 0 OR INPUT_G6_VAR.G6_ERROR2 > 0 THEN
		INPUT_G6_VAR.O_G6_STOP :=TRUE ;			
		TMR10(IN:=INPUT_G6_VAR.O_G6_STOP,PT:=T#1S);
		INPUT_VAR.ALARM1:=INPUT_G6_VAR.I_G6_ERROR OR INPUT_G6_VAR.G6_ERROR1> 0 OR INPUT_G6_VAR.G6_ERROR2 > 0;
		IF NOT TMR10.Q AND INPUT_G6_VAR.I_G6_READY THEN
			INPUT_G6_VAR.O_G6_RESET :=TRUE;	
			INPUT_G6_VAR.O_G6_START :=FALSE ;
			INPUT_G6_VAR.O_G6_CONTINUE :=FALSE;
			INPUT_G6_VAR.O_G6_STOP :=FALSE ;	
			TMR10(IN:=FALSE);
		END_IF
	ELSE
		INPUT_G6_VAR.O_G6_RESET :=FALSE;	
	END_IF
IF INPUT_G6_VAR.I_G6_MOTORON AND NOT INPUT_G6_VAR.I_G6_ESTOPON AND NOT INPUT_G6_VAR.I_G6_SAFEGUARDON AND INDEXING_1_VAR.I_INDEXING_1_ROTATION_DONE  THEN
IF (INPUT_G6_VAR.I_G6_READY OR INPUT_G6_VAR.I_G6_RUNNING) AND NOT INPUT_G6_VAR.I_G6_ERROR AND NOT INPUT_G6_VAR.I_CMDERROR THEN
	
//START FOR 1ST TIME
		IF INPUT_G6_VAR.I_G6_READY  AND NOT INPUT_G6_VAR.I_G6_RUNNING THEN
			INPUT_G6_VAR.O_G6_STOP:=FALSE;
			INPUT_G6_VAR.O_G6_CONTINUE :=FALSE;
			INPUT_G6_VAR.O_G6_PAUSE:=FALSE;
			INPUT_G6_VAR.O_G6_RESET :=FALSE;
			TMR7(IN:=INPUT_G6_VAR.I_G6_READY,PT:=T#1S);
			START_ROBOT(IN:=TMR7.Q,PT:=T#2S);
			INPUT_G6_VAR.O_G6_START :=TMR7.Q ;
		ELSE
			TMR7(IN:=FALSE);
			INPUT_G6_VAR.O_G6_START :=FALSE ;
		END_IF
		IF  NOT INPUT_G6_VAR.I_G6_READY OR INPUT_G6_VAR.I_G6_RUNNING THEN
			INPUT_G6_VAR.O_G6_START :=FALSE ;
		END_IF
		IF INPUT_G6_VAR.I_G6_READY AND INPUT_G6_VAR.O_G6_START THEN
			TMR_HANG(IN:=TRUE,PT:=T#30S);
			IF TMR_HANG.Q THEN
				INPUT_G6_VAR.O_G6_START :=FALSE ;
				INPUT_G6_VAR.O_G6_STOP :=TRUE ;
			END_IF
		ELSE
			TMR_HANG(IN:=FALSE);
		END_IF
//STOP 
		IF INPUT_G6_VAR.I_G6_END_FUKUDA OR( NOT INPUT_G6_VAR.I_G6_READY AND NOT INPUT_G6_VAR.I_G6_RUNNING) THEN
			TMR8(IN:=FALSE);
			TMR9(IN:=FALSE);
		//	INPUT_G6_VAR.O_G6_STOP:=TRUE;
		//	LOADER_RS4_VAR.O_LOADER_RS4_STOP:=TRUE;
		END_IF
		TMR2(IN:=INPUT_G6_VAR.O_G6_STOP,PT:=T#1S);
		IF TMR2.Q THEN
			INPUT_G6_VAR.I_G6_HANG:=FALSE;
			INPUT_G6_VAR.O_G6_STOP:=FALSE;
			TMR1(IN:=FALSE);
		END_IF

		
//CONTINUE	
		//INPUT_G6_VAR.GO_ROBOT:=(INPUT_G6_VAR.I_G6_READY_PLACING AND LOADER_RS4_VAR.I_LOADER_RS4_READY_TAKEUP AND INDEXING_2_VAR.O_ROTATION_DONE )OR(INPUT_G6_VAR.I_G6_READY_PLACING AND NOT LOADER_RS4_VAR.I_LOADER_RS4_ENABLE AND  INDEXING_1_VAR.I_INDEXING_1_ROTATION_DONE)    ;	
		IF (INPUT_G6_VAR.I_G6_READY_PLACING AND LOADER_RS4_VAR.I_LOADER_RS4_READY_TAKEUP AND  INDEXING_1_VAR.I_INDEXING_1_ROTATION_DONE AND INDEXING_2_VAR.I_INDEXING_2_ROTATION_DONE)  THEN
			INPUT_G6_VAR.GO_ROBOT:=TRUE;
		END_IF
		IF (INPUT_G6_VAR.I_G6_READY_PLACING AND NOT LOADER_RS4_VAR.I_LOADER_RS4_ENABLE AND  INDEXING_1_VAR.I_INDEXING_1_ROTATION_DONE AND INDEXING_2_VAR.I_INDEXING_2_ROTATION_DONE) THEN
			INPUT_G6_VAR.GO_ROBOT:=TRUE;
		END_IF
		IF INPUT_G6_VAR.I_G6_START_TAKEUP THEN
			INPUT_G6_VAR.GO_ROBOT:=FALSE;
		END_IF	
		IF INDEXING_1_VAR.I_INDEXING_1_ROTATION_DONE AND INPUT_G6_VAR.GO_ROBOT AND INPUT_VAR.STRAIGHTEN_DONE  AND INPUT_G6_VAR.I_G6_RUNNING AND NOT LOADER_RS4_VAR.I_LOADER_RS4_END_CARRIER THEN
			TMR3(IN:=INPUT_G6_VAR.GO_ROBOT ,PT:=T#0.5S);
			TP1(IN:=INPUT_G6_VAR.GO_ROBOT,PT:=T#0.1S);
		ELSE
			TMR3(IN:=FALSE);
			TP1(IN:=FALSE);
		END_IF
		
		IF INPUT_G6_VAR.I_G6_RUNNING AND  INDEXING_1_VAR.I_INDEXING_1_ROTATION_DONE THEN
			INPUT_G6_VAR.O_G6_START :=FALSE ;
			INPUT_G6_VAR.O_G6_CONTINUE :=TMR3.Q;
			IF (CNT_CYCLE.CV <=3 AND INPUT_G6_VAR.I_G6_READY_TAKEUP AND (INPUT_VAR.I_FUKUDA_TRANSFER_AT_FRONT_A OR INPUT_VAR.I_FUKUDA_TRANSFER_AT_FRONT_B)) AND  INDEXING_1_VAR.I_INDEXING_1_ROTATION_DONE THEN
				INPUT_G6_VAR.O_G6_CONTINUE :=TRUE;
			END_IF
		END_IF
		
//ENABLE ROBOT LOADER RS4
		CNT_CYCLE(CU:=INPUT_G6_VAR.I_G6_START_PLACING,RESET:=NOT INPUT_G6_VAR.I_G6_ENABLE,PV:=4);
		IF CNT_CYCLE.CV =3 AND NOT LOADER_RS4_VAR.I_LOADER_RS4_ENABLE  THEN
			LOADER_RS4_VAR.I_LOADER_RS4_ENABLE:=TRUE;
		END_IF
//PAUSE
		CNT_CYCLE1(CU:=INPUT_G6_VAR.I_G6_START_TAKEUP,RESET:=NOT INPUT_G6_VAR.I_G6_ENABLE,PV:=5);
		IF CNT_CYCLE.CV >=4 AND NOT LOADER_RS4_VAR.I_LOADER_RS4_ENABLE AND  INPUT_G6_VAR.I_G6_RUNNING THEN
			///INPUT_G6_VAR.O_G6_PAUSE:=TRUE;
		END_IF
//START ROTATE INDEXING 1
		IF NOT LOADER_RS4_VAR.I_LOADER_RS4_ENABLE  AND  (INPUT_G6_VAR.IX_G6_GRIPPER_EXT_1 AND INPUT_G6_VAR.I_G6_START_TAKEUP )  THEN
			START_ROTATE(CLK:=TRUE);
			INDEXING_1_VAR.O_ROTATION_START:=TRUE;
		ELSE
			START_ROTATE(CLK:=FALSE);
		END_IF
		IF INPUT_G6_VAR.I_G6_START_PLACING THEN
			INDEXING_1_VAR.O_ROTATION_START:=FALSE;
		END_IF
		
 //SYNCRONIZE ROBOT G6 AND RS4 
		IF INPUT_G6_VAR.I_G6_START_TAKEUP AND LOADER_RS4_VAR.I_LOADER_RS4_START_PLACING  THEN
			INPUT_G6_VAR.GO_ROBOT:=FALSE;
			INPUT_G6_VAR.I_READY_CONTINUE:=FALSE;
			LOADER_RS4_VAR.I_READY_CONTINUE:=FALSE;
		END_IF
		
		IF INPUT_G6_VAR.I_READY_CONTINUE AND LOADER_RS4_VAR.I_READY_CONTINUE THEN
			//INPUT_G6_VAR.O_G6_CONTINUE :=TRUE;
			//LOADER_RS4_VAR.O_LOADER_RS4_CONTINUE :=TRUE;
		END_IF
		
 //END FUKUDA21
 //INPUT_G6_VAR.I_MAX_DEVICE:=40;
// IF INPUT_G6_VAR.I_G6_START_takeup THEN
	 TEMP_COUNTER_FUKUDA_A:=INPUT_G6_VAR.COUNTER_FUKUDA_A;
	 TEMP_COUNTER_FUKUDA_B:=INPUT_G6_VAR.COUNTER_FUKUDA_B;
// END_IF
 		
		IF TEMP_COUNTER_FUKUDA_A >=INPUT_G6_VAR.I_MAX_DEVICE   OR TEMP_COUNTER_FUKUDA_B >=INPUT_G6_VAR.I_MAX_DEVICE THEN
			INPUT_G6_VAR.O_G6_RESET_COUNTER_PICK:=TRUE;
			INPUT_G6_VAR.START_POSITION:=1;
			//TEMP_COUNTER_FUKUDA_A:=0;
			ELSE
				INPUT_G6_VAR.O_G6_RESET_COUNTER_PICK:=FALSE;
		END_IF
		
		IF TEMP_COUNTER_FUKUDA_A >=INPUT_G6_VAR.I_MAX_DEVICE THEN
			O_END_FUKUDA:=TRUE;
			//INPUT_G6_VAR.O_G6_SELECT_FUKUDA_A:=TRUE;
			//INPUT_VAR.I_FUKUDA_TRANSFER_A_PICK_DONE:=TRUE;
			//TEMP_COUNTER_FUKUDA_A:=0;
			ELSE
				O_END_FUKUDA:=FALSE;
		END_IF
		
		IF TEMP_COUNTER_FUKUDA_B >=INPUT_G6_VAR.I_MAX_DEVICE THEN
			O_END_FUKUDB:=TRUE;
			//INPUT_G6_VAR.O_G6_SELECT_FUKUDA_A:=FALSE;
			//INPUT_VAR.I_FUKUDA_TRANSFER_B_PICK_DONE:=TRUE;
			ELSE
			O_END_FUKUDB:=FALSE;
		END_IF

	IF INPUT_G6_VAR.O_G6_GRIPPER_CLOSE_1  THEN
 		GRP1(IN:=TRUE,PT:=T#0.1S);
		ELSE
		GRP1(IN:=FALSE);	
	END_IF
	IF INPUT_G6_VAR.O_G6_GRIPPER_CLOSE_2  THEN
 		GRP2(IN:=TRUE,PT:=T#0.1S); 
		ELSE
		GRP2(IN:=FALSE);	
	END_IF
	IF INPUT_G6_VAR.O_G6_GRIPPER_CLOSE_3  THEN
 		GRP3(IN:=TRUE,PT:=T#0.1S);
		ELSE
		GRP3(IN:=FALSE);	
	END_IF
	IF INPUT_G6_VAR.O_G6_GRIPPER_CLOSE_4  THEN
 		GRP4(IN:=TRUE,PT:=T#0.1S);
		ELSE
		GRP4(IN:=FALSE);	
	END_IF
//	IF LOADER_RS4_VAR.I_LOADER_RS4_START_PLACING THEN
		CNT_TAKING.CU:=(GRP1.Q OR GRP2.Q OR GRP3.Q OR GRP4.Q); 
//	END_IF
	CNT_PLACING(RESET:=INDEXING_2_VAR.O_ROTATION_START,PV:=68);

END_IF
END_IF
ELSE
	//INPUT_G6_VAR.O_G6_STOP :=TRUE ;
	//INPUT_G6_VAR.O_G6_RESET :=TRUE;	
	(*INPUT_G6_VAR.O_G6_START :=FALSE ;
	INPUT_G6_VAR.O_G6_CONTINUE :=FALSE;
	
	INPUT_G6_VAR.O_G6_SETMOTORON:=FALSE;
	
	INPUT_G6_VAR.O_G6_GRIPPER_EXT_DOWN_1:=FALSE;
	INPUT_G6_VAR.O_G6_GRIPPER_EXT_UP_1:=TRUE;
	
	INPUT_G6_VAR.O_G6_GRIPPER_EXT_DOWN_2:=FALSE;
	INPUT_G6_VAR.O_G6_GRIPPER_EXT_UP_2:=TRUE;
	
	INPUT_G6_VAR.O_G6_GRIPPER_EXT_DOWN_3:=FALSE;
	INPUT_G6_VAR.O_G6_GRIPPER_EXT_UP_3:=TRUE;
	
	INPUT_G6_VAR.O_G6_GRIPPER_EXT_DOWN_4:=FALSE;
	INPUT_G6_VAR.O_G6_GRIPPER_EXT_UP_4:=TRUE;
	
	IF INPUT_G6_VAR.I_G6_READY THEN
		INPUT_G6_VAR.O_G6_SETMOTOROFF:=TRUE;
	END_IF
	*)
END_IF
//END_IF

END_PROGRAM

// ---- POUs/ROBOT/TESTER_C8.TcPOU
 PROGRAM TESTER_C8
VAR
	TMR11: TON;
	TMR12: TON;
	TMR10: TON;
	TMR8: TON;
	TMR9: TON;
	TMR7: TON;
	TMR3: TON;
	TP1: TP;
	TMR1: TON;
	START_ROBOT: TP;
	TP2: TP;
	O_G6_HANG: BOOL;
	I_G6_HANG: BOOL;
	TMR2: TON;
	GO_ROBOT: BOOL;
	TP3: TP;
	TMR4: TON;
	CNT_CYCLE: CTU;
	START_ROTATE: R_TRIG;
	IN: INT;
	TMR_RELEASE: TON;
	TMR_OFF_MCAL: TON;
	TMR_RLS_SCAN: TON;
	AFTER_SCAN: BOOL;

	AFTER_SCAN1: BOOL;
	TMR_RLS_SCAN1: TON;
	C8_SEQ: INT;
	DLY1: TON;
	DLY2: TON;
	TMR_RLS: TON;
	TMR_RST: TON;
END_VAR


//GRIPPING CONTROL
IF TESTER_C8_VAR.I_C8_GRIPPER THEN
		TESTER_C8_VAR.O_C8_GRIPPER_CLOSE:=TRUE;
		TESTER_C8_VAR.O_C8_GRIPPER_OPEN:=FALSE;
ELSE
		TESTER_C8_VAR.O_C8_GRIPPER_CLOSE:=FALSE;
		TESTER_C8_VAR.O_C8_GRIPPER_OPEN:=TRUE;
END_IF

IF TESTER_C8_VAR.I_C8_SERROR THEN
	POWER_CONTROL.O_PWR_CTRL_ROBOT_C8:=TRUE;
	TMR_RELEASE(IN:=TRUE,PT:=T#0.5S);
	IF TMR_RELEASE.Q THEN
		POWER_CONTROL.O_PWR_CTRL_ROBOT_C8:=FALSE;
	END_IF
ELSE
	TMR_RELEASE(IN:=FALSE);	
END_IF

//MCAL
	IF TESTER_C8_VAR.I_C8_MCAL_REQUEST THEN
		TESTER_C8_VAR.O_G6_SELROBOT_2:=TRUE;
		IF TESTER_C8_VAR.O_G6_SELROBOT_2 THEN
			DLY1(IN:=TRUE,PT:=T#1S);
			IF DLY1.Q THEN
				TESTER_C8_VAR.O_G6_SETMOTORON:=TRUE;
			END_IF
			IF TESTER_C8_VAR.I_C8_MOTORON THEN
				DLY2(IN:=TRUE,PT:=T#1S);
				IF DLY2.Q THEN
					TESTER_C8_VAR.O_G6_MCAL:=TRUE;
					TMR_OFF_MCAL(IN:=TRUE,PT:=T#2S);	
				END_IF
				IF TMR_OFF_MCAL.Q THEN
					//TESTER_C8_VAR.O_G6_SELROBOT_2:=FALSE;
					//TESTER_C8_VAR.O_G6_MCAL:=FALSE;
				END_IF
			END_IF
		END_IF
	ELSE
		TESTER_C8_VAR.O_G6_SELROBOT_2:=FALSE;
		TESTER_C8_VAR.O_G6_MCAL:=FALSE;
		TMR_OFF_MCAL(IN:=FALSE);
		DLY1(IN:=FALSE);
		DLY2(IN:=FALSE);
	END_IF
	
IF NOT TESTER_C8_VAR.I_C8_MCAL_REQUEST AND TESTER_C8_VAR.C8_ERROR_1 >0 OR (TESTER_C8_VAR.C8_ERROR_2 >0 AND TESTER_C8_VAR.C8_ERROR_2 <32) OR TESTER_C8_VAR.I_C8_ERROR THEN
	TESTER_C8_VAR.O_G6_STOP:=TRUE;
	TMR_RST(IN:=TESTER_C8_VAR.O_G6_STOP,PT:=T#1S);
	IF TMR_RST.Q AND TESTER_C8_VAR.I_C8_READY THEN
		TESTER_C8_VAR.O_G6_STOP:=FALSE;
		TESTER_C8_VAR.O_G6_RESET:=TRUE;
		TMR_RST(IN:=FALSE);
	END_IF
ELSE
	TESTER_C8_VAR.O_G6_RESET:=FALSE;
	IF NOT TESTER_C8_VAR.I_C8_MOTORON THEN
		IF TESTER_C8_VAR.I_C8_READY AND NOT TESTER_C8_VAR.I_C8_ESTOPON AND NOT TESTER_C8_VAR.I_C8_SAFEGUARDON THEN
			TESTER_C8_VAR.O_G6_SETMOTORON:=TRUE;
			TESTER_C8_VAR.O_G6_SETMOTOROFF:=FALSE;	
		END_IF
	ELSE
		TESTER_C8_VAR.O_G6_SETMOTORON:=FALSE;
		TESTER_C8_VAR.O_G6_SETMOTOROFF:=FALSE;
	END_IF 
	IF TESTER_C8_VAR.O_C8_ENABLE AND NOT TESTER_C8_VAR.O_G6_MCAL THEN
		//TESTER_C8_VAR.O_G6_SELROBOT_2:=FALSE;
		IF NOT TESTER_C8_VAR.I_C8_ESTOPON AND NOT TESTER_C8_VAR.I_C8_SAFEGUARDON AND TESTER_C8_VAR.I_C8_READY THEN
			TESTER_C8_VAR.O_G6_SETMOTORON:=TRUE;
			TESTER_C8_VAR.O_G6_SETMOTOROFF:=FALSE;
		END_IF
		

		IF FLAG_VAR.ALLOW_EXECUTE_C8 AND NOT TESTER_C8_VAR.C8_ONDUTY THEN
			TESTER_C8_VAR.C8_START_MOVING:=TRUE;
			IF TESTER_C8_VAR.I_C8_RUNNING THEN
				TESTER_C8_VAR.O_G6_CONTINUE:=TRUE;
			END_IF
			IF TESTER_C8_VAR.I_C8_READY THEN
				TESTER_C8_VAR.O_G6_START:=TRUE;
			END_IF	 
			C8_SEQ:=1;
			ELSE
			TESTER_C8_VAR.O_G6_CONTINUE:=FALSE;
		END_IF
//EXECUTE MOVEMENT	
		IF TESTER_C8_VAR.I_C8_MOTORON AND  TESTER_C8_VAR.C8_START_MOVING AND NOT TESTER_C8_VAR.I_C8_ERROR THEN

			IF TESTER_C8_VAR.I_C8_ROTATE_INDEXING_2  AND NOT LOADER_VAR.I_CARRIER_DETECT_2 THEN
				TESTER_C8_VAR.READY_INDEXING:=TRUE;	
			END_IF
		
			CASE  C8_SEQ OF	
			1:
				FLAG_VAR.ALLOW_EXECUTE_C8:=FALSE;
				TESTER_C8_VAR.C8_MOVEMENT_SOURCE:=TESTER_C8_VAR.C8_MACHINE_POSITION.SOURCE_COORDINATE;
				TESTER_C8_VAR.C8_MOVEMENT_DESTINATION:=TESTER_C8_VAR.C8_MACHINE_POSITION.DESTINATION_COORDINATE;
				C8_SEQ:=2;
				TESTER_C8_VAR.O_G6_FINISH_SCANBARCODE :=FALSE;
			2:
//MOVEMENT TYPE
				IF NOT TESTER_C8_VAR.C8_ONDUTY THEN
					IF TESTER_C8_VAR.C8_MACHINE_POSITION.SOURCE_COORDINATE=0 AND TESTER_C8_VAR.C8_MACHINE_POSITION.DESTINATION_COORDINATE >0 THEN
						TESTER_C8_VAR.C8_PUTON:=TRUE;
						TESTER_C8_VAR.C8_TAKING:=FALSE;
						TESTER_C8_VAR.C8_TRANSFER:=FALSE;
						C8_SEQ:=3;
					END_IF
					 IF TESTER_C8_VAR.C8_MACHINE_POSITION.SOURCE_COORDINATE>0 AND TESTER_C8_VAR.C8_MACHINE_POSITION.DESTINATION_COORDINATE =0 THEN
						TESTER_C8_VAR.C8_PUTON:=FALSE;
						TESTER_C8_VAR.C8_TAKING:=TRUE;
						TESTER_C8_VAR.C8_TRANSFER:=FALSE;
						C8_SEQ:=3;
					END_IF
				 	IF TESTER_C8_VAR.C8_MACHINE_POSITION.SOURCE_COORDINATE>0 AND TESTER_C8_VAR.C8_MACHINE_POSITION.DESTINATION_COORDINATE >0 THEN
						TESTER_C8_VAR.C8_PUTON:=FALSE;
						TESTER_C8_VAR.C8_TAKING:=FALSE;
						TESTER_C8_VAR.C8_TRANSFER:=TRUE;
						C8_SEQ:=3;
					END_IF
				END_IF
3:
//ON DUTY CONTROL
			IF TESTER_C8_VAR.C8_PUTON OR TESTER_C8_VAR.C8_TAKING OR TESTER_C8_VAR.C8_TRANSFER AND NOT TESTER_C8_VAR.I_C8_FREE THEN
				TESTER_C8_VAR.C8_ONDUTY :=TRUE;
			ELSE
				TESTER_C8_VAR.C8_ONDUTY :=FALSE;
			END_IF
//MOVE CARRIER JIG FROM INDEXING TO MACHINE
			IF TESTER_C8_VAR.C8_PUTON THEN
				IF TESTER_C8_VAR.I_C8_READY THEN
					TESTER_C8_VAR.O_G6_START :=TRUE;
					TESTER_C8_VAR.O_G6_CONTINUE :=FALSE;
				ELSE
					TESTER_C8_VAR.O_G6_START :=FALSE;
				END_IF
				
				(*IF TESTER_C8_VAR.I_C8_READY_SCAN THEN
					TESTER_C8_VAR.O_G6_FINISH_SCANBARCODE :=TRUE;
					AFTER_SCAN:=TRUE ;
				END_IF*)
				//TESTER_C8_VAR.O_G6_FINISH_SCANBARCODE :=TESTER_C8_VAR.I_C8_READY_SCAN;
				IF TESTER_C8_VAR.O_G6_FINISH_SCANBARCODE THEN
					AFTER_SCAN:=TRUE;
				END_IF
				IF TESTER_C8_VAR.I_C8_RUNNING  AND NOT AFTER_SCAN AND NOT TESTER_C8_VAR.I_C8_FREE THEN
					TESTER_C8_VAR.O_G6_START :=FALSE;
				//	TESTER_C8_VAR.O_G6_CONTINUE :=TRUE;
				END_IF
				
				TMR_RLS_SCAN(IN:=AFTER_SCAN,PT:=T#1S);
				IF TMR_RLS_SCAN.Q THEN
						TESTER_C8_VAR.O_G6_FINISH_SCANBARCODE :=FALSE;
						TESTER_C8_VAR.O_G6_CONTINUE :=FALSE;
						TESTER_C8_VAR.C8_PUTON:=FALSE;
						AFTER_SCAN:=FALSE;
						TMR_RLS_SCAN(IN:=FALSE);
						C8_SEQ:=4;
						
